Yaskawa INFORM job: DEMO_ROOF_UPPER_0625_3PAINT_41.JBI

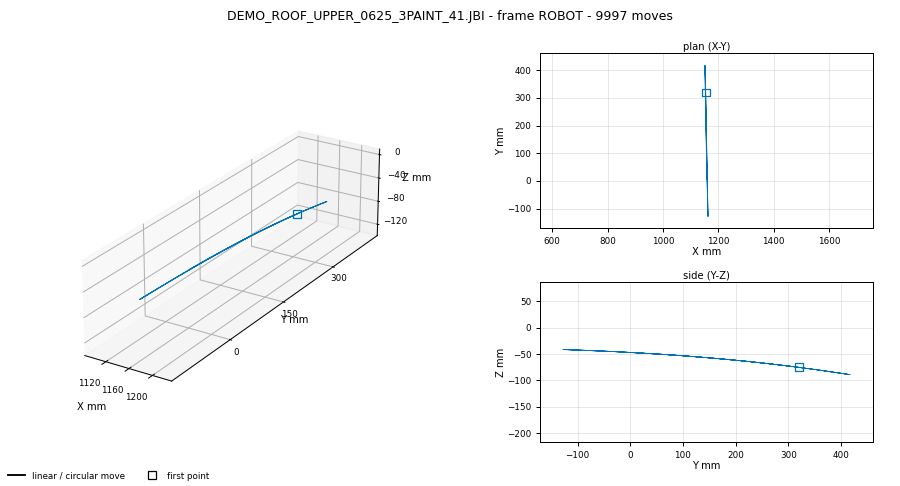
[picture p0: tool path of DEMO_ROOF_UPPER_0625_3PAINT_41.JBI in frame ROBOT, 9997 of 9997 moves have a stored position in this frame; points joined in program order, loops and branches not executed]
/JOB
//NAME DEMO_ROOF_UPPER_0625_3PAINT41
//POS
///NPOS 9997,0,0,0,0,0
///TOOL 0
///USER 0
///POSTYPE ROBOT
///RECTAN
///RCONF 1,0,0,0,0,0,0,0,0,0,0,0,0,0,0,0,0,0,0,0,0,0,0,0
C00000=1155.027,319.870,-75.171,-176.725,8.570,148.744
C00001=1155.032,319.622,-75.138,-176.728,8.567,148.744
C00002=1155.036,319.374,-75.107,-176.730,8.563,148.743
C00003=1155.040,319.126,-75.075,-176.733,8.560,148.743
C00004=1155.044,318.878,-75.042,-176.735,8.557,148.743
C00005=1155.048,318.630,-75.011,-176.738,8.553,148.743
C00006=1155.052,318.382,-74.979,-176.741,8.550,148.743
C00007=1155.057,318.134,-74.947,-176.743,8.546,148.743
C00008=1155.060,317.886,-74.915,-176.746,8.542,148.742
C00009=1155.065,317.639,-74.883,-176.748,8.539,148.742
C00010=1155.069,317.390,-74.851,-176.751,8.536,148.742
C00011=1155.073,317.142,-74.819,-176.753,8.533,148.742
C00012=1155.077,316.895,-74.788,-176.756,8.529,148.742
C00013=1155.081,316.647,-74.756,-176.758,8.525,148.742
C00014=1155.085,316.399,-74.723,-176.761,8.522,148.742
C00015=1155.090,316.151,-74.692,-176.764,8.519,148.742
C00016=1155.093,315.903,-74.660,-176.766,8.515,148.741
C00017=1155.097,315.655,-74.629,-176.769,8.512,148.741
C00018=1155.102,315.407,-74.597,-176.771,8.509,148.741
C00019=1155.106,315.159,-74.565,-176.774,8.506,148.741
C00020=1155.110,314.911,-74.533,-176.777,8.502,148.741
C00021=1155.114,314.663,-74.502,-176.779,8.499,148.741
C00022=1155.119,314.415,-74.469,-176.782,8.495,148.741
C00023=1155.123,314.167,-74.438,-176.784,8.492,148.740
C00024=1155.128,313.890,-74.403,-176.787,8.488,148.740
C00025=1155.132,313.612,-74.367,-176.790,8.484,148.740
C00026=1155.137,313.335,-74.332,-176.793,8.480,148.740
C00027=1155.141,313.058,-74.296,-176.795,8.477,148.740
C00028=1155.146,312.810,-74.265,-176.799,8.473,148.740
C00029=1155.149,312.562,-74.234,-176.801,8.470,148.739
C00030=1155.153,312.314,-74.202,-176.803,8.466,148.739
C00031=1155.159,312.065,-74.170,-176.806,8.463,148.739
C00032=1155.162,311.817,-74.139,-176.809,8.460,148.739
C00033=1155.167,311.570,-74.107,-176.811,8.456,148.739
C00034=1155.171,311.321,-74.076,-176.814,8.453,148.739
C00035=1155.175,311.074,-74.045,-176.816,8.450,148.739
C00036=1155.179,310.826,-74.013,-176.819,8.447,148.739
C00037=1155.183,310.578,-73.982,-176.822,8.443,148.739
C00038=1155.187,310.330,-73.950,-176.824,8.440,148.738
C00039=1155.191,310.082,-73.919,-176.827,8.436,148.738
C00040=1155.195,309.834,-73.887,-176.830,8.433,148.738
C00041=1155.200,309.586,-73.857,-176.832,8.430,148.738
C00042=1155.204,309.338,-73.825,-176.835,8.426,148.738
C00043=1155.208,309.090,-73.794,-176.837,8.423,148.738
C00044=1155.212,308.842,-73.762,-176.840,8.420,148.738
C00045=1155.216,308.594,-73.731,-176.842,8.416,148.737
C00046=1155.220,308.346,-73.700,-176.845,8.413,148.737
C00047=1155.225,308.098,-73.669,-176.848,8.409,148.737
C00048=1155.228,307.850,-73.637,-176.850,8.406,148.737
C00049=1155.233,307.602,-73.606,-176.853,8.403,148.737
C00050=1155.237,307.353,-73.575,-176.855,8.400,148.737
C00051=1155.241,307.106,-73.544,-176.858,8.397,148.737
C00052=1155.245,306.857,-73.513,-176.861,8.393,148.737
C00053=1155.250,306.610,-73.481,-176.863,8.389,148.736
C00054=1155.254,306.362,-73.450,-176.866,8.387,148.737
C00055=1155.258,306.114,-73.419,-176.868,8.383,148.736
C00056=1155.263,305.866,-73.388,-176.871,8.380,148.736
C00057=1155.267,305.618,-73.357,-176.874,8.376,148.736
C00058=1155.271,305.370,-73.326,-176.876,8.373,148.736
C00059=1155.275,305.121,-73.295,-176.879,8.370,148.736
C00060=1155.279,304.874,-73.264,-176.881,8.367,148.736
C00061=1155.283,304.626,-73.233,-176.884,8.364,148.736
C00062=1155.287,304.377,-73.202,-176.887,8.360,148.736
C00063=1155.292,304.129,-73.171,-176.889,8.356,148.735
C00064=1155.296,303.882,-73.140,-176.892,8.353,148.735
C00065=1155.300,303.633,-73.108,-176.894,8.350,148.735
C00066=1155.304,303.386,-73.078,-176.897,8.347,148.735
C00067=1155.308,303.137,-73.047,-176.899,8.344,148.735
C00068=1155.313,302.889,-73.016,-176.903,8.340,148.735
C00069=1155.317,302.642,-72.985,-176.905,8.337,148.735
C00070=1155.321,302.393,-72.954,-176.907,8.334,148.735
C00071=1155.325,302.145,-72.924,-176.910,8.331,148.735
C00072=1155.330,301.897,-72.893,-176.912,8.327,148.735
C00073=1155.334,301.649,-72.862,-176.915,8.324,148.735
C00074=1155.338,301.401,-72.831,-176.918,8.320,148.734
C00075=1155.342,301.153,-72.801,-176.921,8.317,148.734
C00076=1155.346,300.905,-72.770,-176.923,8.314,148.734
C00077=1155.351,300.657,-72.739,-176.926,8.311,148.734
C00078=1155.355,300.409,-72.708,-176.928,8.308,148.734
C00079=1155.359,300.161,-72.678,-176.931,8.305,148.734
C00080=1155.363,299.912,-72.647,-176.934,8.301,148.734
C00081=1155.368,299.664,-72.616,-176.937,8.298,148.734
C00082=1155.372,299.417,-72.586,-176.939,8.295,148.734
C00083=1155.376,299.168,-72.555,-176.941,8.291,148.734
C00084=1155.380,298.920,-72.524,-176.944,8.288,148.734
C00085=1155.384,298.672,-72.494,-176.946,8.285,148.733
C00086=1155.389,298.424,-72.463,-176.950,8.281,148.733
C00087=1155.393,298.176,-72.432,-176.952,8.278,148.733
C00088=1155.397,297.928,-72.402,-176.955,8.275,148.733
C00089=1155.402,297.680,-72.372,-176.957,8.272,148.733
C00090=1155.406,297.432,-72.342,-176.960,8.269,148.733
C00091=1155.410,297.183,-72.310,-176.962,8.266,148.733
C00092=1155.414,296.935,-72.280,-176.965,8.263,148.733
C00093=1155.418,296.688,-72.250,-176.968,8.259,148.733
C00094=1155.423,296.440,-72.219,-176.970,8.255,148.733
C00095=1155.426,296.191,-72.189,-176.973,8.253,148.733
C00096=1155.431,295.943,-72.158,-176.976,8.249,148.733
C00097=1155.435,295.695,-72.128,-176.978,8.246,148.733
C00098=1155.439,295.447,-72.097,-176.981,8.243,148.733
C00099=1155.444,295.199,-72.068,-176.983,8.240,148.733
C00100=1155.448,294.950,-72.037,-176.986,8.237,148.732
C00101=1155.452,294.703,-72.006,-176.989,8.233,148.732
C00102=1155.456,294.454,-71.976,-176.991,8.230,148.732
C00103=1155.460,294.206,-71.946,-176.994,8.227,148.732
C00104=1155.465,293.958,-71.916,-176.996,8.224,148.732
C00105=1155.468,293.709,-71.886,-176.999,8.221,148.732
C00106=1155.473,293.461,-71.855,-177.002,8.218,148.732
C00107=1155.477,293.214,-71.825,-177.004,8.214,148.732
C00108=1155.482,292.965,-71.795,-177.007,8.211,148.732
C00109=1155.486,292.718,-71.765,-177.010,8.207,148.732
C00110=1155.490,292.469,-71.735,-177.013,8.204,148.732
C00111=1155.495,292.221,-71.704,-177.015,8.201,148.732
C00112=1155.498,291.973,-71.674,-177.018,8.198,148.732
C00113=1155.503,291.724,-71.644,-177.020,8.195,148.732
C00114=1155.507,291.477,-71.614,-177.023,8.192,148.732
C00115=1155.511,291.229,-71.584,-177.026,8.189,148.732
C00116=1155.515,290.981,-71.553,-177.028,8.186,148.731
C00117=1155.520,290.732,-71.524,-177.031,8.183,148.731
C00118=1155.523,290.485,-71.494,-177.033,8.179,148.731
C00119=1155.528,290.236,-71.464,-177.036,8.176,148.731
C00120=1155.533,289.988,-71.434,-177.039,8.173,148.731
C00121=1155.536,289.739,-71.404,-177.041,8.169,148.731
C00122=1155.541,289.491,-71.374,-177.044,8.166,148.731
C00123=1155.545,289.243,-71.343,-177.046,8.163,148.731
C00124=1155.549,288.995,-71.314,-177.049,8.160,148.731
C00125=1155.554,288.746,-71.284,-177.052,8.157,148.731
C00126=1155.558,288.499,-71.254,-177.054,8.154,148.731
C00127=1155.562,288.251,-71.224,-177.057,8.151,148.731
C00128=1155.566,287.976,-71.191,-177.060,8.147,148.731
C00129=1155.571,287.700,-71.158,-177.063,8.144,148.731
C00130=1155.576,287.426,-71.125,-177.066,8.140,148.731
C00131=1155.580,287.149,-71.092,-177.069,8.137,148.731
C00132=1155.585,286.902,-71.061,-177.072,8.133,148.731
C00133=1155.589,286.653,-71.032,-177.074,8.130,148.731
C00134=1155.593,286.405,-71.002,-177.077,8.127,148.731
C00135=1155.598,286.157,-70.973,-177.080,8.124,148.731
C00136=1155.602,285.909,-70.942,-177.082,8.121,148.731
C00137=1155.606,285.661,-70.913,-177.085,8.118,148.731
C00138=1155.611,285.412,-70.883,-177.087,8.115,148.730
C00139=1155.615,285.164,-70.854,-177.090,8.112,148.730
C00140=1155.619,284.916,-70.825,-177.093,8.109,148.731
C00141=1155.624,284.668,-70.795,-177.095,8.106,148.730
C00142=1155.628,284.420,-70.765,-177.098,8.103,148.730
C00143=1155.632,284.172,-70.735,-177.101,8.100,148.730
C00144=1155.637,283.924,-70.706,-177.103,8.096,148.730
C00145=1155.641,283.675,-70.676,-177.106,8.094,148.730
C00146=1155.645,283.427,-70.647,-177.109,8.091,148.730
C00147=1155.649,283.179,-70.617,-177.111,8.086,148.730
C00148=1155.653,282.931,-70.588,-177.114,8.084,148.730
C00149=1155.658,282.682,-70.558,-177.117,8.081,148.730
C00150=1155.662,282.434,-70.529,-177.119,8.077,148.730
C00151=1155.666,282.186,-70.500,-177.122,8.074,148.730
C00152=1155.671,281.937,-70.469,-177.125,8.071,148.730
C00153=1155.675,281.689,-70.440,-177.128,8.068,148.730
C00154=1155.679,281.441,-70.411,-177.130,8.065,148.730
C00155=1155.684,281.193,-70.381,-177.133,8.062,148.730
C00156=1155.688,280.945,-70.352,-177.135,8.059,148.730
C00157=1155.692,280.697,-70.323,-177.138,8.056,148.730
C00158=1155.697,280.448,-70.293,-177.140,8.053,148.730
C00159=1155.701,280.200,-70.264,-177.143,8.050,148.730
C00160=1155.705,279.952,-70.234,-177.146,8.047,148.730
C00161=1155.709,279.703,-70.205,-177.148,8.044,148.730
C00162=1155.714,279.455,-70.176,-177.151,8.041,148.730
C00163=1155.718,279.207,-70.147,-177.154,8.038,148.730
C00164=1155.722,278.959,-70.118,-177.157,8.035,148.730
C00165=1155.726,278.711,-70.089,-177.159,8.032,148.730
C00166=1155.730,278.463,-70.059,-177.162,8.029,148.730
C00167=1155.735,278.214,-70.030,-177.164,8.026,148.730
C00168=1155.739,277.965,-70.001,-177.167,8.023,148.730
C00169=1155.744,277.718,-69.972,-177.170,8.020,148.730
C00170=1155.748,277.470,-69.942,-177.172,8.017,148.730
C00171=1155.752,277.221,-69.914,-177.175,8.014,148.730
C00172=1155.756,276.972,-69.884,-177.178,8.010,148.730
C00173=1155.761,276.724,-69.855,-177.181,8.007,148.730
C00174=1155.765,276.477,-69.826,-177.184,8.004,148.730
C00175=1155.769,276.228,-69.798,-177.186,8.001,148.730
C00176=1155.773,275.980,-69.768,-177.189,7.998,148.730
C00177=1155.778,275.731,-69.739,-177.191,7.995,148.730
C00178=1155.782,275.483,-69.710,-177.194,7.992,148.730
C00179=1155.787,275.235,-69.681,-177.197,7.989,148.730
C00180=1155.790,274.987,-69.652,-177.200,7.986,148.730
C00181=1155.795,274.738,-69.623,-177.202,7.983,148.730
C00182=1155.799,274.490,-69.594,-177.205,7.979,148.730
C00183=1155.804,274.242,-69.565,-177.207,7.977,148.730
C00184=1155.807,273.994,-69.537,-177.210,7.974,148.730
C00185=1155.812,273.745,-69.508,-177.213,7.971,148.730
C00186=1155.816,273.497,-69.478,-177.216,7.968,148.730
C00187=1155.821,273.248,-69.450,-177.218,7.964,148.730
C00188=1155.825,273.000,-69.421,-177.221,7.961,148.730
C00189=1155.829,272.752,-69.392,-177.224,7.959,148.730
C00190=1155.833,272.503,-69.363,-177.226,7.956,148.730
C00191=1155.838,272.255,-69.335,-177.229,7.953,148.730
C00192=1155.842,272.007,-69.306,-177.231,7.949,148.730
C00193=1155.846,271.758,-69.277,-177.234,7.946,148.730
C00194=1155.851,271.511,-69.248,-177.237,7.943,148.730
C00195=1155.855,271.262,-69.220,-177.240,7.941,148.730
C00196=1155.859,271.014,-69.190,-177.243,7.938,148.730
C00197=1155.864,270.766,-69.162,-177.245,7.935,148.730
C00198=1155.868,270.517,-69.134,-177.248,7.931,148.730
C00199=1155.872,270.269,-69.104,-177.250,7.928,148.730
C00200=1155.877,270.021,-69.076,-177.253,7.926,148.730
C00201=1155.881,269.772,-69.048,-177.255,7.923,148.730
C00202=1155.885,269.524,-69.018,-177.258,7.920,148.730
C00203=1155.890,269.276,-68.990,-177.261,7.917,148.730
C00204=1155.894,269.027,-68.962,-177.263,7.914,148.730
C00205=1155.899,268.779,-68.933,-177.266,7.911,148.730
C00206=1155.902,268.531,-68.905,-177.269,7.908,148.730
C00207=1155.907,268.282,-68.876,-177.272,7.905,148.730
C00208=1155.911,268.034,-68.848,-177.274,7.902,148.730
C00209=1155.916,267.785,-68.819,-177.277,7.899,148.730
C00210=1155.920,267.537,-68.790,-177.280,7.896,148.730
C00211=1155.924,267.289,-68.762,-177.283,7.894,148.731
C00212=1155.929,267.040,-68.733,-177.285,7.890,148.730
C00213=1155.933,266.792,-68.706,-177.288,7.887,148.730
C00214=1155.938,266.543,-68.677,-177.290,7.884,148.730
C00215=1155.942,266.296,-68.648,-177.293,7.881,148.731
C00216=1155.946,266.047,-68.620,-177.296,7.878,148.731
C00217=1155.950,265.799,-68.591,-177.299,7.876,148.731
C00218=1155.955,265.551,-68.563,-177.302,7.873,148.731
C00219=1155.959,265.302,-68.535,-177.304,7.870,148.731
C00220=1155.964,265.054,-68.507,-177.307,7.867,148.731
C00221=1155.968,264.805,-68.478,-177.309,7.863,148.731
C00222=1155.973,264.557,-68.450,-177.312,7.860,148.731
C00223=1155.976,264.308,-68.422,-177.315,7.858,148.731
C00224=1155.981,264.061,-68.394,-177.318,7.855,148.731
C00225=1155.985,263.812,-68.365,-177.320,7.852,148.731
C00226=1155.990,263.564,-68.338,-177.323,7.850,148.731
C00227=1155.994,263.315,-68.309,-177.325,7.847,148.731
C00228=1155.998,263.067,-68.281,-177.328,7.844,148.731
C00229=1156.002,262.818,-68.253,-177.331,7.841,148.731
C00230=1156.007,262.570,-68.225,-177.334,7.838,148.731
C00231=1156.011,262.322,-68.196,-177.336,7.835,148.731
C00232=1156.016,262.048,-68.166,-177.339,7.832,148.731
C00233=1156.021,261.775,-68.135,-177.343,7.828,148.731
C00234=1156.026,261.501,-68.104,-177.345,7.825,148.731
C00235=1156.030,261.229,-68.072,-177.348,7.822,148.731
C00236=1156.035,260.980,-68.045,-177.351,7.819,148.732
C00237=1156.039,260.731,-68.017,-177.354,7.816,148.732
C00238=1156.044,260.483,-67.989,-177.356,7.813,148.732
C00239=1156.047,260.235,-67.961,-177.359,7.810,148.732
C00240=1156.052,259.987,-67.933,-177.362,7.807,148.732
C00241=1156.057,259.738,-67.905,-177.365,7.805,148.732
C00242=1156.061,259.490,-67.877,-177.368,7.802,148.732
C00243=1156.065,259.242,-67.849,-177.370,7.798,148.732
C00244=1156.069,258.993,-67.821,-177.373,7.795,148.732
C00245=1156.074,258.745,-67.793,-177.375,7.792,148.732
C00246=1156.078,258.496,-67.765,-177.378,7.790,148.732
C00247=1156.082,258.248,-67.738,-177.380,7.787,148.732
C00248=1156.087,258.000,-67.710,-177.383,7.784,148.732
C00249=1156.092,257.750,-67.682,-177.386,7.781,148.732
C00250=1156.096,257.503,-67.654,-177.389,7.779,148.732
C00251=1156.100,257.254,-67.626,-177.391,7.776,148.732
C00252=1156.104,257.006,-67.599,-177.394,7.773,148.732
C00253=1156.109,256.758,-67.571,-177.397,7.770,148.732
C00254=1156.113,256.509,-67.542,-177.400,7.767,148.732
C00255=1156.118,256.260,-67.515,-177.403,7.764,148.732
C00256=1156.122,256.012,-67.488,-177.405,7.762,148.733
C00257=1156.126,255.763,-67.460,-177.407,7.759,148.733
C00258=1156.131,255.515,-67.432,-177.410,7.756,148.733
C00259=1156.135,255.267,-67.405,-177.413,7.753,148.733
C00260=1156.139,255.018,-67.377,-177.416,7.750,148.733
C00261=1156.144,254.770,-67.350,-177.419,7.747,148.733
C00262=1156.149,254.522,-67.322,-177.421,7.744,148.733
C00263=1156.153,254.273,-67.294,-177.424,7.741,148.733
C00264=1156.157,254.025,-67.266,-177.427,7.738,148.733
C00265=1156.162,253.776,-67.239,-177.429,7.736,148.733
C00266=1156.166,253.527,-67.211,-177.432,7.733,148.733
C00267=1156.170,253.279,-67.184,-177.435,7.730,148.734
C00268=1156.175,253.031,-67.156,-177.438,7.728,148.734
C00269=1156.179,252.783,-67.129,-177.441,7.725,148.734
C00270=1156.183,252.534,-67.101,-177.443,7.722,148.734
C00271=1156.188,252.286,-67.074,-177.446,7.719,148.734
C00272=1156.192,252.037,-67.047,-177.449,7.716,148.734
C00273=1156.196,251.788,-67.019,-177.451,7.714,148.734
C00274=1156.201,251.540,-66.992,-177.454,7.711,148.734
C00275=1156.205,251.291,-66.965,-177.457,7.708,148.734
C00276=1156.210,251.044,-66.937,-177.459,7.705,148.734
C00277=1156.214,250.794,-66.910,-177.462,7.702,148.734
C00278=1156.218,250.546,-66.883,-177.465,7.699,148.734
C00279=1156.223,250.298,-66.855,-177.468,7.696,148.734
C00280=1156.227,250.050,-66.828,-177.470,7.694,148.734
C00281=1156.232,249.800,-66.800,-177.473,7.691,148.735
C00282=1156.236,249.552,-66.773,-177.476,7.688,148.735
C00283=1156.240,249.304,-66.746,-177.478,7.685,148.735
C00284=1156.244,249.056,-66.719,-177.482,7.682,148.735
C00285=1156.249,248.807,-66.692,-177.484,7.680,148.735
C00286=1156.253,248.558,-66.665,-177.487,7.677,148.735
C00287=1156.258,248.310,-66.637,-177.489,7.674,148.735
C00288=1156.262,248.062,-66.610,-177.492,7.672,148.735
C00289=1156.267,247.813,-66.583,-177.495,7.669,148.735
C00290=1156.271,247.565,-66.556,-177.498,7.666,148.735
C00291=1156.275,247.317,-66.529,-177.500,7.663,148.735
C00292=1156.279,247.067,-66.502,-177.503,7.660,148.736
C00293=1156.284,246.819,-66.475,-177.505,7.658,148.736
C00294=1156.289,246.570,-66.448,-177.508,7.655,148.736
C00295=1156.293,246.322,-66.420,-177.511,7.652,148.736
C00296=1156.298,246.073,-66.393,-177.514,7.649,148.736
C00297=1156.302,245.826,-66.366,-177.517,7.646,148.736
C00298=1156.306,245.577,-66.339,-177.520,7.643,148.736
C00299=1156.310,245.328,-66.312,-177.522,7.641,148.736
C00300=1156.315,245.080,-66.285,-177.525,7.638,148.736
C00301=1156.319,244.831,-66.258,-177.527,7.635,148.736
C00302=1156.324,244.583,-66.231,-177.530,7.632,148.737
C00303=1156.328,244.334,-66.204,-177.533,7.630,148.737
C00304=1156.333,244.086,-66.177,-177.536,7.628,148.737
C00305=1156.337,243.837,-66.151,-177.538,7.625,148.737
C00306=1156.342,243.589,-66.124,-177.541,7.622,148.737
C00307=1156.346,243.340,-66.097,-177.544,7.619,148.737
C00308=1156.350,243.091,-66.070,-177.547,7.616,148.737
C00309=1156.354,242.843,-66.043,-177.549,7.614,148.737
C00310=1156.359,242.594,-66.016,-177.552,7.611,148.737
C00311=1156.364,242.346,-65.989,-177.555,7.608,148.738
C00312=1156.368,242.098,-65.963,-177.558,7.605,148.738
C00313=1156.372,241.849,-65.936,-177.560,7.602,148.738
C00314=1156.377,241.600,-65.910,-177.563,7.600,148.738
C00315=1156.381,241.352,-65.883,-177.565,7.597,148.738
C00316=1156.386,241.103,-65.856,-177.568,7.594,148.738
C00317=1156.390,240.855,-65.829,-177.571,7.592,148.738
C00318=1156.394,240.607,-65.802,-177.574,7.589,148.738
C00319=1156.399,240.357,-65.776,-177.576,7.587,148.739
C00320=1156.403,240.109,-65.749,-177.579,7.584,148.739
C00321=1156.408,239.861,-65.722,-177.582,7.581,148.739
C00322=1156.412,239.612,-65.697,-177.585,7.578,148.739
C00323=1156.417,239.363,-65.670,-177.588,7.575,148.739
C00324=1156.422,239.115,-65.642,-177.590,7.573,148.739
C00325=1156.425,238.867,-65.616,-177.593,7.570,148.739
C00326=1156.430,238.618,-65.590,-177.596,7.567,148.739
C00327=1156.434,238.370,-65.563,-177.599,7.564,148.739
C00328=1156.439,238.121,-65.536,-177.601,7.563,148.740
C00329=1156.443,237.872,-65.510,-177.604,7.560,148.740
C00330=1156.448,237.624,-65.483,-177.607,7.557,148.740
C00331=1156.452,237.375,-65.458,-177.610,7.554,148.740
C00332=1156.457,237.126,-65.431,-177.612,7.552,148.740
C00333=1156.461,236.878,-65.404,-177.615,7.549,148.740
C00334=1156.466,236.629,-65.378,-177.618,7.546,148.740
C00335=1156.470,236.381,-65.351,-177.621,7.543,148.741
C00336=1156.475,236.109,-65.323,-177.623,7.540,148.741
C00337=1156.479,235.837,-65.294,-177.627,7.538,148.741
C00338=1156.484,235.566,-65.264,-177.629,7.535,148.741
C00339=1156.489,235.294,-65.236,-177.632,7.532,148.741
C00340=1156.494,235.045,-65.209,-177.635,7.529,148.741
C00341=1156.498,234.797,-65.184,-177.638,7.526,148.741
C00342=1156.502,234.548,-65.157,-177.640,7.524,148.742
C00343=1156.507,234.299,-65.131,-177.643,7.521,148.742
C00344=1156.512,234.051,-65.105,-177.646,7.518,148.742
C00345=1156.516,233.803,-65.078,-177.649,7.516,148.742
C00346=1156.521,233.554,-65.053,-177.651,7.514,148.742
C00347=1156.525,233.306,-65.026,-177.654,7.511,148.742
C00348=1156.530,233.057,-65.000,-177.657,7.508,148.742
C00349=1156.534,232.808,-64.974,-177.660,7.505,148.743
C00350=1156.538,232.560,-64.948,-177.662,7.503,148.743
C00351=1156.543,232.311,-64.921,-177.665,7.500,148.743
C00352=1156.547,232.062,-64.896,-177.668,7.497,148.743
C00353=1156.551,231.814,-64.869,-177.671,7.494,148.743
C00354=1156.556,231.565,-64.843,-177.673,7.492,148.743
C00355=1156.561,231.316,-64.817,-177.676,7.489,148.743
C00356=1156.564,231.068,-64.791,-177.679,7.486,148.743
C00357=1156.570,230.820,-64.765,-177.682,7.485,148.744
C00358=1156.574,230.571,-64.739,-177.684,7.482,148.744
C00359=1156.579,230.322,-64.713,-177.687,7.479,148.744
C00360=1156.582,230.074,-64.687,-177.690,7.476,148.744
C00361=1156.587,229.825,-64.661,-177.693,7.474,148.744
C00362=1156.592,229.576,-64.635,-177.695,7.471,148.744
C00363=1156.596,229.328,-64.609,-177.698,7.468,148.744
C00364=1156.601,229.079,-64.584,-177.701,7.466,148.745
C00365=1156.605,228.830,-64.558,-177.704,7.464,148.745
C00366=1156.610,228.582,-64.531,-177.706,7.461,148.745
C00367=1156.614,228.334,-64.505,-177.709,7.458,148.745
C00368=1156.619,228.085,-64.480,-177.712,7.456,148.745
C00369=1156.623,227.836,-64.454,-177.715,7.453,148.745
C00370=1156.627,227.587,-64.428,-177.717,7.450,148.746
C00371=1156.633,227.339,-64.402,-177.720,7.448,148.746
C00372=1156.637,227.090,-64.376,-177.723,7.445,148.746
C00373=1156.641,226.841,-64.351,-177.726,7.442,148.746
C00374=1156.645,226.592,-64.325,-177.728,7.441,148.746
C00375=1156.650,226.344,-64.300,-177.731,7.438,148.746
C00376=1156.654,226.096,-64.274,-177.734,7.435,148.747
C00377=1156.659,225.847,-64.248,-177.736,7.433,148.747
C00378=1156.663,225.599,-64.223,-177.739,7.430,148.747
C00379=1156.668,225.350,-64.196,-177.742,7.427,148.747
C00380=1156.673,225.101,-64.171,-177.744,7.425,148.747
C00381=1156.677,224.852,-64.145,-177.747,7.422,148.747
C00382=1156.682,224.604,-64.119,-177.750,7.419,148.748
C00383=1156.686,224.355,-64.094,-177.752,7.417,148.748
C00384=1156.690,224.106,-64.068,-177.756,7.415,148.748
C00385=1156.695,223.858,-64.043,-177.758,7.412,148.748
C00386=1156.699,223.609,-64.017,-177.761,7.410,148.748
C00387=1156.703,223.360,-63.991,-177.764,7.407,148.749
C00388=1156.708,223.112,-63.966,-177.767,7.404,148.749
C00389=1156.713,222.863,-63.941,-177.769,7.402,148.749
C00390=1156.717,222.614,-63.915,-177.772,7.399,148.749
C00391=1156.722,222.366,-63.890,-177.775,7.397,148.749
C00392=1156.726,222.117,-63.864,-177.777,7.394,148.749
C00393=1156.731,221.869,-63.838,-177.780,7.392,148.750
C00394=1156.735,221.620,-63.813,-177.783,7.389,148.750
C00395=1156.740,221.371,-63.788,-177.786,7.387,148.750
C00396=1156.744,221.123,-63.762,-177.789,7.384,148.750
C00397=1156.749,220.874,-63.736,-177.791,7.381,148.750
C00398=1156.753,220.625,-63.711,-177.794,7.380,148.750
C00399=1156.758,220.376,-63.686,-177.797,7.377,148.751
C00400=1156.762,220.128,-63.660,-177.799,7.374,148.751
C00401=1156.766,219.880,-63.635,-177.802,7.372,148.751
C00402=1156.771,219.630,-63.610,-177.805,7.369,148.751
C00403=1156.775,219.382,-63.585,-177.807,7.367,148.751
C00404=1156.780,219.134,-63.559,-177.811,7.364,148.751
C00405=1156.784,218.884,-63.534,-177.813,7.361,148.752
C00406=1156.789,218.636,-63.509,-177.816,7.360,148.752
C00407=1156.793,218.387,-63.483,-177.819,7.357,148.752
C00408=1156.799,218.138,-63.458,-177.821,7.355,148.752
C00409=1156.802,217.890,-63.433,-177.824,7.352,148.752
C00410=1156.807,217.641,-63.409,-177.827,7.349,148.753
C00411=1156.811,217.392,-63.383,-177.829,7.347,148.753
C00412=1156.816,217.144,-63.357,-177.832,7.344,148.753
C00413=1156.821,216.895,-63.332,-177.835,7.341,148.753
C00414=1156.824,216.646,-63.307,-177.838,7.340,148.753
C00415=1156.829,216.398,-63.283,-177.841,7.337,148.753
C00416=1156.834,216.149,-63.257,-177.843,7.335,148.754
C00417=1156.839,215.900,-63.232,-177.846,7.332,148.754
C00418=1156.843,215.651,-63.206,-177.849,7.329,148.754
C00419=1156.847,215.403,-63.182,-177.852,7.327,148.754
C00420=1156.852,215.154,-63.157,-177.854,7.324,148.754
C00421=1156.857,214.905,-63.132,-177.857,7.322,148.755
C00422=1156.861,214.656,-63.108,-177.860,7.320,148.755
C00423=1156.865,214.408,-63.082,-177.862,7.318,148.755
C00424=1156.870,214.159,-63.057,-177.865,7.315,148.755
C00425=1156.875,213.911,-63.032,-177.868,7.312,148.755
C00426=1156.879,213.662,-63.008,-177.871,7.310,148.756
C00427=1156.884,213.413,-62.983,-177.874,7.307,148.756
C00428=1156.888,213.165,-62.957,-177.876,7.305,148.756
C00429=1156.892,212.916,-62.933,-177.879,7.303,148.756
C00430=1156.897,212.668,-62.907,-177.882,7.300,148.756
C00431=1156.902,212.418,-62.882,-177.885,7.298,148.757
C00432=1156.906,212.170,-62.858,-177.887,7.295,148.757
C00433=1156.911,211.920,-62.833,-177.890,7.293,148.757
C00434=1156.915,211.672,-62.808,-177.893,7.290,148.757
C00435=1156.920,211.424,-62.784,-177.895,7.288,148.757
C00436=1156.924,211.174,-62.759,-177.898,7.286,148.758
C00437=1156.928,210.927,-62.734,-177.900,7.283,148.758
C00438=1156.933,210.677,-62.709,-177.904,7.281,148.758
C00439=1156.938,210.428,-62.684,-177.906,7.278,148.758
C00440=1156.943,210.158,-62.658,-177.909,7.276,148.759
C00441=1156.948,209.887,-62.631,-177.912,7.273,148.759
C00442=1156.953,209.617,-62.604,-177.915,7.271,148.759
C00443=1156.957,209.346,-62.577,-177.918,7.268,148.759
C00444=1156.962,209.098,-62.553,-177.921,7.265,148.759
C00445=1156.967,208.849,-62.528,-177.924,7.263,148.760
C00446=1156.971,208.600,-62.504,-177.927,7.261,148.760
C00447=1156.976,208.351,-62.479,-177.929,7.259,148.760
C00448=1156.980,208.102,-62.454,-177.932,7.256,148.760
C00449=1156.985,207.853,-62.430,-177.934,7.254,148.760
C00450=1156.990,207.605,-62.404,-177.938,7.251,148.761
C00451=1156.993,207.356,-62.380,-177.940,7.249,148.761
C00452=1156.999,207.108,-62.355,-177.943,7.246,148.761
C00453=1157.003,206.859,-62.331,-177.945,7.244,148.761
C00454=1157.007,206.611,-62.307,-177.949,7.242,148.762
C00455=1157.012,206.361,-62.282,-177.951,7.239,148.762
C00456=1157.016,206.113,-62.258,-177.954,7.237,148.762
C00457=1157.021,205.864,-62.233,-177.957,7.234,148.762
C00458=1157.025,205.615,-62.209,-177.959,7.232,148.763
C00459=1157.030,205.366,-62.184,-177.962,7.229,148.763
C00460=1157.035,205.118,-62.160,-177.965,7.228,148.763
C00461=1157.040,204.869,-62.135,-177.968,7.225,148.763
C00462=1157.044,204.620,-62.111,-177.970,7.223,148.763
C00463=1157.048,204.371,-62.088,-177.973,7.220,148.764
C00464=1157.053,204.122,-62.063,-177.976,7.218,148.764
C00465=1157.057,203.873,-62.039,-177.979,7.215,148.764
C00466=1157.062,203.625,-62.014,-177.981,7.214,148.764
C00467=1157.067,203.376,-61.990,-177.984,7.211,148.764
C00468=1157.071,203.128,-61.966,-177.987,7.209,148.765
C00469=1157.075,202.879,-61.941,-177.990,7.206,148.765
C00470=1157.080,202.630,-61.917,-177.992,7.204,148.765
C00471=1157.085,202.381,-61.893,-177.995,7.202,148.766
C00472=1157.089,202.132,-61.869,-177.998,7.200,148.766
C00473=1157.094,201.884,-61.845,-178.001,7.197,148.766
C00474=1157.098,201.635,-61.820,-178.003,7.195,148.766
C00475=1157.103,201.386,-61.796,-178.006,7.192,148.766
C00476=1157.108,201.137,-61.772,-178.009,7.190,148.767
C00477=1157.112,200.888,-61.748,-178.012,7.188,148.767
C00478=1157.117,200.640,-61.724,-178.014,7.185,148.767
C00479=1157.121,200.391,-61.699,-178.017,7.183,148.767
C00480=1157.126,200.141,-61.676,-178.020,7.181,148.767
C00481=1157.130,199.893,-61.651,-178.023,7.178,148.768
C00482=1157.135,199.645,-61.627,-178.025,7.176,148.768
C00483=1157.139,199.396,-61.604,-178.028,7.174,148.768
C00484=1157.145,199.147,-61.579,-178.031,7.172,148.769
C00485=1157.148,198.898,-61.555,-178.033,7.170,148.769
C00486=1157.153,198.649,-61.532,-178.036,7.167,148.769
C00487=1157.157,198.400,-61.507,-178.039,7.165,148.769
C00488=1157.162,198.152,-61.483,-178.042,7.162,148.770
C00489=1157.167,197.903,-61.459,-178.044,7.160,148.770
C00490=1157.172,197.654,-61.435,-178.047,7.158,148.770
C00491=1157.176,197.405,-61.412,-178.050,7.156,148.770
C00492=1157.180,197.156,-61.388,-178.053,7.153,148.770
C00493=1157.185,196.907,-61.364,-178.056,7.151,148.771
C00494=1157.189,196.659,-61.340,-178.058,7.148,148.771
C00495=1157.194,196.410,-61.317,-178.061,7.147,148.771
C00496=1157.199,196.161,-61.292,-178.063,7.145,148.771
C00497=1157.204,195.912,-61.269,-178.066,7.142,148.772
C00498=1157.208,195.663,-61.245,-178.069,7.140,148.772
C00499=1157.213,195.414,-61.221,-178.072,7.137,148.772
C00500=1157.217,195.166,-61.197,-178.075,7.135,148.773
C00501=1157.222,194.917,-61.174,-178.077,7.133,148.773
C00502=1157.226,194.669,-61.150,-178.080,7.131,148.773
C00503=1157.231,194.419,-61.126,-178.083,7.128,148.773
C00504=1157.235,194.170,-61.102,-178.086,7.126,148.773
C00505=1157.240,193.921,-61.079,-178.088,7.124,148.774
C00506=1157.244,193.672,-61.055,-178.091,7.121,148.774
C00507=1157.249,193.424,-61.031,-178.094,7.120,148.774
C00508=1157.253,193.175,-61.008,-178.097,7.117,148.775
C00509=1157.258,192.926,-60.984,-178.099,7.115,148.775
C00510=1157.262,192.677,-60.960,-178.102,7.112,148.775
C00511=1157.267,192.428,-60.937,-178.105,7.110,148.775
C00512=1157.272,192.180,-60.913,-178.107,7.109,148.776
C00513=1157.276,191.931,-60.890,-178.111,7.106,148.776
C00514=1157.281,191.682,-60.866,-178.113,7.104,148.776
C00515=1157.286,191.433,-60.843,-178.116,7.101,148.776
C00516=1157.290,191.184,-60.819,-178.119,7.100,148.777
C00517=1157.295,190.935,-60.795,-178.121,7.097,148.777
C00518=1157.299,190.686,-60.772,-178.124,7.095,148.777
C00519=1157.304,190.437,-60.749,-178.126,7.093,148.777
C00520=1157.309,190.189,-60.725,-178.130,7.090,148.778
C00521=1157.313,189.940,-60.701,-178.132,7.088,148.778
C00522=1157.318,189.691,-60.678,-178.135,7.086,148.778
C00523=1157.323,189.442,-60.655,-178.138,7.084,148.778
C00524=1157.327,189.193,-60.631,-178.141,7.082,148.779
C00525=1157.332,188.944,-60.607,-178.143,7.079,148.779
C00526=1157.337,188.696,-60.584,-178.146,7.077,148.779
C00527=1157.341,188.447,-60.561,-178.149,7.076,148.780
C00528=1157.346,188.198,-60.538,-178.152,7.073,148.780
C00529=1157.350,187.949,-60.515,-178.154,7.071,148.780
C00530=1157.355,187.700,-60.491,-178.158,7.068,148.780
C00531=1157.360,187.451,-60.468,-178.160,7.066,148.781
C00532=1157.365,187.202,-60.445,-178.162,7.065,148.781
C00533=1157.369,186.953,-60.421,-178.166,7.062,148.781
C00534=1157.373,186.704,-60.399,-178.168,7.060,148.781
C00535=1157.378,186.456,-60.374,-178.171,7.057,148.782
C00536=1157.382,186.207,-60.351,-178.174,7.056,148.782
C00537=1157.387,185.958,-60.328,-178.176,7.053,148.782
C00538=1157.392,185.710,-60.305,-178.179,7.051,148.783
C00539=1157.396,185.461,-60.282,-178.182,7.049,148.783
C00540=1157.401,185.212,-60.259,-178.184,7.047,148.783
C00541=1157.406,184.963,-60.235,-178.187,7.044,148.783
C00542=1157.411,184.713,-60.213,-178.190,7.043,148.784
C00543=1157.415,184.464,-60.190,-178.192,7.041,148.784
C00544=1157.420,184.195,-60.164,-178.196,7.038,148.784
C00545=1157.425,183.926,-60.139,-178.199,7.035,148.785
C00546=1157.430,183.656,-60.115,-178.202,7.034,148.785
C00547=1157.435,183.386,-60.090,-178.205,7.031,148.785
C00548=1157.440,183.137,-60.066,-178.207,7.029,148.785
C00549=1157.444,182.888,-60.043,-178.210,7.026,148.786
C00550=1157.448,182.640,-60.020,-178.213,7.025,148.786
C00551=1157.454,182.391,-59.997,-178.215,7.023,148.786
C00552=1157.459,182.142,-59.974,-178.219,7.020,148.787
C00553=1157.462,181.893,-59.952,-178.221,7.018,148.787
C00554=1157.467,181.644,-59.928,-178.224,7.017,148.787
C00555=1157.471,181.395,-59.906,-178.227,7.014,148.787
C00556=1157.476,181.147,-59.883,-178.229,7.012,148.788
C00557=1157.481,180.897,-59.860,-178.232,7.010,148.788
C00558=1157.485,180.648,-59.837,-178.235,7.007,148.788
C00559=1157.490,180.399,-59.814,-178.238,7.005,148.789
C00560=1157.495,180.150,-59.790,-178.240,7.004,148.789
C00561=1157.500,179.902,-59.769,-178.244,7.001,148.789
C00562=1157.504,179.653,-59.745,-178.246,6.999,148.789
C00563=1157.508,179.404,-59.723,-178.248,6.997,148.790
C00564=1157.513,179.154,-59.700,-178.252,6.995,148.790
C00565=1157.518,178.906,-59.678,-178.254,6.993,148.790
C00566=1157.523,178.657,-59.654,-178.257,6.991,148.791
C00567=1157.527,178.408,-59.632,-178.260,6.988,148.791
C00568=1157.532,178.159,-59.609,-178.263,6.987,148.791
C00569=1157.537,177.911,-59.586,-178.265,6.984,148.792
C00570=1157.541,177.661,-59.564,-178.268,6.982,148.792
C00571=1157.546,177.412,-59.540,-178.271,6.980,148.792
C00572=1157.550,177.164,-59.518,-178.273,6.978,148.793
C00573=1157.555,176.914,-59.495,-178.276,6.975,148.793
C00574=1157.559,176.666,-59.473,-178.279,6.974,148.793
C00575=1157.564,176.416,-59.450,-178.282,6.972,148.793
C00576=1157.569,176.168,-59.428,-178.284,6.970,148.794
C00577=1157.574,175.918,-59.405,-178.287,6.967,148.794
C00578=1157.578,175.670,-59.382,-178.290,6.966,148.794
C00579=1157.583,175.421,-59.361,-178.292,6.964,148.795
C00580=1157.587,175.172,-59.337,-178.296,6.961,148.795
C00581=1157.592,174.923,-59.315,-178.298,6.959,148.795
C00582=1157.597,174.674,-59.292,-178.301,6.957,148.796
C00583=1157.601,174.425,-59.270,-178.304,6.955,148.796
C00584=1157.606,174.176,-59.247,-178.307,6.953,148.796
C00585=1157.611,173.927,-59.225,-178.309,6.951,148.797
C00586=1157.615,173.679,-59.202,-178.312,6.949,148.797
C00587=1157.620,173.429,-59.180,-178.315,6.947,148.797
C00588=1157.624,173.181,-59.157,-178.317,6.945,148.797
C00589=1157.629,172.931,-59.135,-178.320,6.943,148.798
C00590=1157.634,172.683,-59.113,-178.322,6.941,148.798
C00591=1157.638,172.434,-59.090,-178.326,6.939,148.798
C00592=1157.643,172.184,-59.067,-178.328,6.937,148.799
C00593=1157.648,171.936,-59.046,-178.331,6.935,148.799
C00594=1157.652,171.687,-59.023,-178.334,6.933,148.799
C00595=1157.658,171.438,-59.001,-178.337,6.930,148.800
C00596=1157.662,171.189,-58.979,-178.339,6.929,148.800
C00597=1157.666,170.940,-58.956,-178.342,6.927,148.800
C00598=1157.672,170.691,-58.934,-178.345,6.924,148.801
C00599=1157.676,170.442,-58.912,-178.348,6.923,148.801
C00600=1157.681,170.193,-58.890,-178.350,6.921,148.801
C00601=1157.685,169.944,-58.867,-178.353,6.919,148.802
C00602=1157.690,169.695,-58.845,-178.356,6.916,148.802
C00603=1157.695,169.446,-58.823,-178.359,6.914,148.802
C00604=1157.699,169.197,-58.801,-178.361,6.913,148.803
C00605=1157.704,168.948,-58.778,-178.364,6.911,148.803
C00606=1157.708,168.699,-58.756,-178.367,6.908,148.803
C00607=1157.713,168.450,-58.734,-178.370,6.906,148.804
C00608=1157.717,168.201,-58.712,-178.372,6.905,148.804
C00609=1157.722,167.952,-58.690,-178.375,6.903,148.804
C00610=1157.727,167.703,-58.668,-178.378,6.900,148.804
C00611=1157.732,167.455,-58.645,-178.381,6.898,148.805
C00612=1157.736,167.205,-58.623,-178.383,6.896,148.805
C00613=1157.741,166.957,-58.602,-178.386,6.895,148.805
C00614=1157.745,166.707,-58.580,-178.389,6.893,148.806
C00615=1157.751,166.458,-58.557,-178.392,6.890,148.806
C00616=1157.755,166.209,-58.535,-178.394,6.888,148.806
C00617=1157.760,165.960,-58.514,-178.397,6.887,148.807
C00618=1157.764,165.711,-58.491,-178.400,6.885,148.807
C00619=1157.769,165.462,-58.470,-178.403,6.882,148.807
C00620=1157.773,165.213,-58.448,-178.405,6.881,148.808
C00621=1157.778,164.964,-58.426,-178.408,6.879,148.808
C00622=1157.783,164.715,-58.403,-178.410,6.877,148.808
C00623=1157.788,164.466,-58.382,-178.413,6.875,148.809
C00624=1157.793,164.218,-58.360,-178.416,6.872,148.809
C00625=1157.797,163.968,-58.338,-178.419,6.871,148.809
C00626=1157.802,163.720,-58.316,-178.422,6.869,148.810
C00627=1157.806,163.470,-58.294,-178.424,6.867,148.810
C00628=1157.811,163.222,-58.273,-178.427,6.865,148.811
C00629=1157.816,162.972,-58.251,-178.430,6.863,148.811
C00630=1157.821,162.724,-58.229,-178.433,6.861,148.811
C00631=1157.825,162.475,-58.207,-178.435,6.859,148.811
C00632=1157.830,162.226,-58.185,-178.438,6.857,148.812
C00633=1157.835,161.977,-58.163,-178.441,6.856,148.812
C00634=1157.839,161.728,-58.141,-178.444,6.853,148.813
C00635=1157.844,161.478,-58.120,-178.447,6.851,148.813
C00636=1157.848,161.229,-58.098,-178.449,6.850,148.813
C00637=1157.853,160.980,-58.077,-178.452,6.847,148.813
C00638=1157.858,160.732,-58.055,-178.454,6.846,148.814
C00639=1157.862,160.482,-58.033,-178.458,6.843,148.814
C00640=1157.867,160.234,-58.011,-178.460,6.841,148.815
C00641=1157.872,159.984,-57.990,-178.463,6.840,148.815
C00642=1157.877,159.735,-57.968,-178.466,6.838,148.815
C00643=1157.881,159.487,-57.947,-178.468,6.836,148.816
C00644=1157.886,159.238,-57.925,-178.471,6.834,148.816
C00645=1157.891,158.988,-57.904,-178.474,6.832,148.816
C00646=1157.896,158.739,-57.882,-178.477,6.830,148.817
C00647=1157.900,158.490,-57.860,-178.479,6.828,148.817
C00648=1157.905,158.222,-57.837,-178.482,6.826,148.817
C00649=1157.911,157.952,-57.814,-178.485,6.824,148.818
C00650=1157.915,157.684,-57.791,-178.488,6.822,148.818
C00651=1157.921,157.414,-57.767,-178.491,6.820,148.818
C00652=1157.925,157.165,-57.745,-178.494,6.818,148.819
C00653=1157.930,156.916,-57.724,-178.497,6.816,148.819
C00654=1157.934,156.667,-57.703,-178.499,6.814,148.820
C00655=1157.939,156.419,-57.681,-178.502,6.813,148.820
C00656=1157.944,156.169,-57.660,-178.505,6.811,148.820
C00657=1157.949,155.920,-57.638,-178.508,6.808,148.821
C00658=1157.954,155.671,-57.617,-178.511,6.807,148.821
C00659=1157.958,155.422,-57.595,-178.513,6.805,148.821
C00660=1157.962,155.173,-57.574,-178.516,6.803,148.822
C00661=1157.967,154.924,-57.553,-178.519,6.801,148.822
C00662=1157.972,154.675,-57.532,-178.521,6.799,148.822
C00663=1157.977,154.425,-57.510,-178.524,6.798,148.823
C00664=1157.982,154.177,-57.489,-178.527,6.795,148.823
C00665=1157.986,153.928,-57.468,-178.530,6.793,148.823
C00666=1157.991,153.679,-57.447,-178.532,6.792,148.824
C00667=1157.996,153.429,-57.425,-178.535,6.790,148.824
C00668=1158.000,153.181,-57.404,-178.538,6.788,148.825
C00669=1158.006,152.931,-57.383,-178.541,6.786,148.825
C00670=1158.010,152.683,-57.362,-178.543,6.785,148.825
C00671=1158.015,152.434,-57.341,-178.546,6.783,148.826
C00672=1158.019,152.184,-57.319,-178.549,6.780,148.826
C00673=1158.024,151.935,-57.298,-178.552,6.779,148.826
C00674=1158.029,151.686,-57.277,-178.555,6.777,148.827
C00675=1158.034,151.438,-57.256,-178.557,6.775,148.827
C00676=1158.039,151.188,-57.235,-178.560,6.773,148.828
C00677=1158.043,150.939,-57.214,-178.562,6.771,148.828
C00678=1158.048,150.690,-57.192,-178.565,6.770,148.828
C00679=1158.053,150.441,-57.171,-178.568,6.768,148.829
C00680=1158.057,150.192,-57.151,-178.570,6.766,148.829
C00681=1158.062,149.943,-57.129,-178.574,6.764,148.829
C00682=1158.067,149.694,-57.108,-178.576,6.762,148.830
C00683=1158.071,149.444,-57.087,-178.579,6.760,148.830
C00684=1158.076,149.196,-57.066,-178.582,6.758,148.830
C00685=1158.081,148.946,-57.045,-178.584,6.757,148.831
C00686=1158.086,148.697,-57.024,-178.587,6.755,148.831
C00687=1158.090,148.449,-57.003,-178.590,6.753,148.832
C00688=1158.095,148.200,-56.982,-178.593,6.751,148.832
C00689=1158.100,147.951,-56.961,-178.595,6.750,148.832
C00690=1158.105,147.701,-56.940,-178.598,6.748,148.833
C00691=1158.109,147.452,-56.920,-178.601,6.745,148.833
C00692=1158.114,147.203,-56.898,-178.604,6.744,148.833
C00693=1158.118,146.954,-56.878,-178.607,6.742,148.834
C00694=1158.123,146.705,-56.857,-178.609,6.740,148.834
C00695=1158.128,146.456,-56.836,-178.612,6.739,148.835
C00696=1158.133,146.207,-56.815,-178.615,6.737,148.835
C00697=1158.137,145.958,-56.794,-178.618,6.735,148.835
C00698=1158.142,145.709,-56.773,-178.620,6.733,148.836
C00699=1158.148,145.460,-56.752,-178.623,6.732,148.836
C00700=1158.151,145.210,-56.732,-178.626,6.730,148.837
C00701=1158.157,144.961,-56.711,-178.628,6.728,148.837
C00702=1158.161,144.712,-56.690,-178.631,6.726,148.837
C00703=1158.166,144.463,-56.669,-178.634,6.725,148.838
C00704=1158.171,144.214,-56.649,-178.636,6.723,148.838
C00705=1158.175,143.965,-56.628,-178.640,6.720,148.838
C00706=1158.180,143.715,-56.608,-178.642,6.719,148.839
C00707=1158.185,143.467,-56.587,-178.645,6.717,148.839
C00708=1158.190,143.217,-56.566,-178.648,6.715,148.840
C00709=1158.194,142.968,-56.546,-178.651,6.713,148.840
C00710=1158.199,142.719,-56.525,-178.653,6.712,148.840
C00711=1158.204,142.470,-56.504,-178.656,6.710,148.841
C00712=1158.208,142.221,-56.484,-178.659,6.708,148.841
C00713=1158.214,141.972,-56.463,-178.661,6.707,148.842
C00714=1158.218,141.723,-56.443,-178.664,6.705,148.842
C00715=1158.223,141.474,-56.422,-178.667,6.703,148.842
C00716=1158.228,141.225,-56.401,-178.669,6.701,148.843
C00717=1158.232,140.976,-56.381,-178.672,6.700,148.843
C00718=1158.237,140.727,-56.360,-178.675,6.698,148.843
C00719=1158.242,140.478,-56.340,-178.678,6.696,148.844
C00720=1158.247,140.228,-56.319,-178.680,6.695,148.844
C00721=1158.251,139.979,-56.298,-178.683,6.693,148.845
C00722=1158.256,139.730,-56.278,-178.686,6.691,148.845
C00723=1158.261,139.481,-56.258,-178.688,6.689,148.845
C00724=1158.266,139.232,-56.237,-178.691,6.688,148.846
C00725=1158.270,138.983,-56.217,-178.694,6.686,148.846
C00726=1158.275,138.733,-56.196,-178.697,6.684,148.847
C00727=1158.280,138.484,-56.176,-178.699,6.682,148.847
C00728=1158.284,138.236,-56.155,-178.702,6.681,148.847
C00729=1158.289,137.986,-56.136,-178.705,6.679,148.848
C00730=1158.294,137.737,-56.115,-178.707,6.677,148.848
C00731=1158.298,137.488,-56.094,-178.710,6.676,148.849
C00732=1158.303,137.239,-56.074,-178.713,6.674,148.849
C00733=1158.308,136.990,-56.055,-178.716,6.672,148.849
C00734=1158.313,136.741,-56.034,-178.718,6.670,148.850
C00735=1158.318,136.492,-56.013,-178.721,6.669,148.850
C00736=1158.322,136.243,-55.993,-178.724,6.667,148.851
C00737=1158.327,135.993,-55.973,-178.727,6.666,148.851
C00738=1158.332,135.744,-55.952,-178.730,6.664,148.852
C00739=1158.337,135.495,-55.932,-178.732,6.662,148.852
C00740=1158.341,135.245,-55.912,-178.735,6.660,148.852
C00741=1158.346,134.996,-55.892,-178.738,6.659,148.853
C00742=1158.352,134.748,-55.871,-178.740,6.657,148.853
C00743=1158.356,134.498,-55.852,-178.743,6.655,148.853
C00744=1158.361,134.249,-55.831,-178.746,6.653,148.854
C00745=1158.366,134.000,-55.812,-178.748,6.652,148.854
C00746=1158.370,133.751,-55.791,-178.751,6.650,148.855
C00747=1158.374,133.502,-55.771,-178.754,6.648,148.855
C00748=1158.380,133.252,-55.751,-178.757,6.647,148.855
C00749=1158.385,133.004,-55.731,-178.759,6.645,148.856
C00750=1158.390,132.754,-55.711,-178.762,6.643,148.856
C00751=1158.394,132.505,-55.691,-178.765,6.641,148.857
C00752=1158.399,132.237,-55.670,-178.768,6.640,148.857
C00753=1158.404,131.968,-55.647,-178.771,6.638,148.858
C00754=1158.409,131.700,-55.626,-178.774,6.636,148.858
C00755=1158.415,131.431,-55.604,-178.777,6.634,148.858
C00756=1158.419,131.182,-55.584,-178.779,6.632,148.859
C00757=1158.424,130.932,-55.564,-178.783,6.631,148.859
C00758=1158.429,130.684,-55.544,-178.785,6.629,148.860
C00759=1158.434,130.434,-55.525,-178.788,6.628,148.860
C00760=1158.438,130.185,-55.504,-178.791,6.626,148.861
C00761=1158.443,129.936,-55.485,-178.793,6.624,148.861
C00762=1158.448,129.687,-55.465,-178.796,6.622,148.861
C00763=1158.453,129.438,-55.445,-178.799,6.621,148.862
C00764=1158.458,129.188,-55.425,-178.802,6.619,148.862
C00765=1158.462,128.940,-55.405,-178.804,6.617,148.863
C00766=1158.467,128.691,-55.386,-178.807,6.616,148.863
C00767=1158.472,128.441,-55.366,-178.810,6.614,148.863
C00768=1158.477,128.192,-55.346,-178.813,6.612,148.864
C00769=1158.481,127.943,-55.326,-178.815,6.612,148.864
C00770=1158.487,127.694,-55.307,-178.818,6.610,148.865
C00771=1158.491,127.445,-55.286,-178.820,6.608,148.865
C00772=1158.496,127.195,-55.267,-178.823,6.606,148.866
C00773=1158.501,126.946,-55.247,-178.826,6.605,148.866
C00774=1158.506,126.697,-55.227,-178.829,6.603,148.866
C00775=1158.510,126.448,-55.207,-178.831,6.601,148.867
C00776=1158.515,126.198,-55.188,-178.834,6.600,148.867
C00777=1158.520,125.949,-55.168,-178.837,6.598,148.868
C00778=1158.525,125.700,-55.148,-178.840,6.596,148.868
C00779=1158.530,125.451,-55.128,-178.843,6.595,148.869
C00780=1158.534,125.201,-55.109,-178.845,6.593,148.869
C00781=1158.540,124.952,-55.089,-178.848,6.591,148.869
C00782=1158.543,124.704,-55.070,-178.851,6.590,148.870
C00783=1158.548,124.454,-55.050,-178.853,6.589,148.870
C00784=1158.553,124.205,-55.031,-178.856,6.587,148.871
C00785=1158.558,123.956,-55.011,-178.859,6.586,148.871
C00786=1158.563,123.706,-54.991,-178.861,6.584,148.872
C00787=1158.568,123.457,-54.972,-178.864,6.582,148.872
C00788=1158.573,123.208,-54.952,-178.867,6.580,148.872
C00789=1158.577,122.959,-54.933,-178.870,6.579,148.873
C00790=1158.582,122.710,-54.913,-178.872,6.577,148.873
C00791=1158.587,122.461,-54.894,-178.875,6.575,148.874
C00792=1158.592,122.211,-54.874,-178.878,6.574,148.874
C00793=1158.597,121.962,-54.855,-178.881,6.572,148.875
C00794=1158.602,121.713,-54.835,-178.883,6.571,148.875
C00795=1158.606,121.464,-54.816,-178.886,6.570,148.875
C00796=1158.611,121.215,-54.797,-178.889,6.568,148.876
C00797=1158.616,120.965,-54.777,-178.891,6.566,148.876
C00798=1158.621,120.716,-54.758,-178.894,6.565,148.877
C00799=1158.625,120.467,-54.739,-178.897,6.563,148.877
C00800=1158.630,120.218,-54.719,-178.900,6.561,148.878
C00801=1158.635,119.968,-54.700,-178.903,6.560,148.878
C00802=1158.640,119.719,-54.680,-178.905,6.558,148.878
C00803=1158.645,119.470,-54.661,-178.907,6.557,148.879
C00804=1158.649,119.221,-54.642,-178.910,6.555,148.879
C00805=1158.655,118.972,-54.622,-178.913,6.554,148.880
C00806=1158.659,118.722,-54.603,-178.916,6.552,148.880
C00807=1158.664,118.474,-54.584,-178.919,6.551,148.881
C00808=1158.669,118.224,-54.564,-178.922,6.549,148.881
C00809=1158.673,117.975,-54.545,-178.924,6.547,148.881
C00810=1158.678,117.726,-54.526,-178.927,6.546,148.882
C00811=1158.683,117.476,-54.506,-178.929,6.545,148.882
C00812=1158.688,117.228,-54.487,-178.932,6.543,148.883
C00813=1158.692,116.978,-54.468,-178.935,6.542,148.883
C00814=1158.698,116.729,-54.450,-178.938,6.540,148.884
C00815=1158.703,116.479,-54.430,-178.940,6.538,148.884
C00816=1158.707,116.231,-54.411,-178.943,6.536,148.885
C00817=1158.712,115.981,-54.392,-178.946,6.535,148.885
C00818=1158.717,115.732,-54.372,-178.948,6.534,148.886
C00819=1158.721,115.483,-54.353,-178.951,6.532,148.886
C00820=1158.727,115.234,-54.335,-178.954,6.531,148.886
C00821=1158.732,114.984,-54.315,-178.957,6.529,148.887
C00822=1158.736,114.735,-54.296,-178.959,6.527,148.887
C00823=1158.741,114.486,-54.277,-178.962,6.526,148.888
C00824=1158.746,114.237,-54.259,-178.965,6.525,148.888
C00825=1158.751,113.987,-54.239,-178.967,6.523,148.889
C00826=1158.755,113.739,-54.220,-178.970,6.522,148.889
C00827=1158.760,113.489,-54.201,-178.973,6.520,148.889
C00828=1158.766,113.240,-54.182,-178.976,6.518,148.890
C00829=1158.770,112.990,-54.163,-178.979,6.517,148.890
C00830=1158.775,112.741,-54.144,-178.981,6.515,148.891
C00831=1158.780,112.492,-54.126,-178.984,6.514,148.891
C00832=1158.785,112.243,-54.106,-178.986,6.513,148.892
C00833=1158.789,111.994,-54.087,-178.989,6.511,148.892
C00834=1158.794,111.744,-54.068,-178.992,6.510,148.893
C00835=1158.799,111.495,-54.050,-178.995,6.508,148.893
C00836=1158.804,111.246,-54.030,-178.997,6.507,148.894
C00837=1158.809,110.997,-54.012,-179.000,6.505,148.894
C00838=1158.814,110.748,-53.993,-179.003,6.504,148.894
C00839=1158.818,110.498,-53.974,-179.006,6.502,148.895
C00840=1158.824,110.249,-53.955,-179.008,6.500,148.895
C00841=1158.828,110.000,-53.936,-179.011,6.499,148.896
C00842=1158.833,109.750,-53.918,-179.013,6.498,148.896
C00843=1158.838,109.502,-53.899,-179.016,6.496,148.897
C00844=1158.843,109.251,-53.880,-179.019,6.495,148.897
C00845=1158.847,109.003,-53.861,-179.022,6.493,148.898
C00846=1158.852,108.753,-53.843,-179.025,6.491,148.898
C00847=1158.857,108.504,-53.824,-179.027,6.491,148.898
C00848=1158.862,108.255,-53.806,-179.030,6.489,148.899
C00849=1158.867,108.005,-53.786,-179.033,6.487,148.900
C00850=1158.872,107.756,-53.768,-179.035,6.486,148.900
C00851=1158.876,107.508,-53.749,-179.038,6.484,148.900
C00852=1158.881,107.258,-53.730,-179.040,6.483,148.901
C00853=1158.886,107.009,-53.712,-179.044,6.482,148.901
C00854=1158.892,106.759,-53.693,-179.046,6.480,148.902
C00855=1158.896,106.510,-53.674,-179.049,6.478,148.902
C00856=1158.901,106.242,-53.655,-179.052,6.477,148.903
C00857=1158.907,105.973,-53.635,-179.055,6.475,148.903
C00858=1158.911,105.706,-53.614,-179.058,6.474,148.904
C00859=1158.917,105.437,-53.594,-179.061,6.472,148.904
C00860=1158.921,105.187,-53.576,-179.063,6.471,148.905
C00861=1158.927,104.938,-53.557,-179.066,6.470,148.905
C00862=1158.931,104.689,-53.538,-179.068,6.468,148.906
C00863=1158.936,104.439,-53.520,-179.072,6.467,148.906
C00864=1158.941,104.191,-53.502,-179.074,6.465,148.907
C00865=1158.946,103.941,-53.483,-179.076,6.464,148.907
C00866=1158.951,103.691,-53.465,-179.079,6.462,148.907
C00867=1158.955,103.442,-53.447,-179.082,6.461,148.908
C00868=1158.961,103.193,-53.428,-179.085,6.459,148.908
C00869=1158.965,102.944,-53.409,-179.087,6.458,148.909
C00870=1158.970,102.694,-53.391,-179.090,6.457,148.909
C00871=1158.975,102.446,-53.373,-179.093,6.455,148.910
C00872=1158.980,102.196,-53.354,-179.096,6.454,148.910
C00873=1158.985,101.946,-53.336,-179.098,6.453,148.911
C00874=1158.990,101.697,-53.318,-179.101,6.451,148.911
C00875=1158.994,101.448,-53.300,-179.104,6.450,148.912
C00876=1158.999,101.200,-53.281,-179.107,6.448,148.912
C00877=1159.004,100.949,-53.262,-179.109,6.447,148.913
C00878=1159.009,100.700,-53.244,-179.112,6.445,148.913
C00879=1159.014,100.451,-53.226,-179.115,6.444,148.914
C00880=1159.019,100.202,-53.208,-179.117,6.442,148.914
C00881=1159.023,99.953,-53.189,-179.120,6.442,148.915
C00882=1159.028,99.703,-53.170,-179.122,6.440,148.915
C00883=1159.033,99.454,-53.152,-179.126,6.439,148.916
C00884=1159.038,99.205,-53.135,-179.128,6.437,148.916
C00885=1159.043,98.956,-53.117,-179.130,6.436,148.916
C00886=1159.048,98.706,-53.099,-179.134,6.435,148.917
C00887=1159.052,98.457,-53.080,-179.136,6.433,148.917
C00888=1159.057,98.207,-53.062,-179.139,6.431,148.918
C00889=1159.063,97.958,-53.044,-179.141,6.430,148.918
C00890=1159.068,97.709,-53.026,-179.144,6.429,148.919
C00891=1159.073,97.460,-53.007,-179.147,6.427,148.919
C00892=1159.077,97.211,-52.989,-179.149,6.426,148.920
C00893=1159.082,96.961,-52.971,-179.152,6.425,148.920
C00894=1159.087,96.712,-52.953,-179.155,6.423,148.921
C00895=1159.092,96.463,-52.935,-179.158,6.422,148.921
C00896=1159.096,96.214,-52.917,-179.160,6.421,148.922
C00897=1159.101,95.964,-52.899,-179.163,6.419,148.922
C00898=1159.106,95.715,-52.881,-179.166,6.418,148.923
C00899=1159.111,95.466,-52.863,-179.168,6.417,148.923
C00900=1159.116,95.216,-52.845,-179.171,6.415,148.924
C00901=1159.121,94.966,-52.827,-179.174,6.414,148.924
C00902=1159.126,94.717,-52.809,-179.177,6.412,148.925
C00903=1159.131,94.468,-52.791,-179.179,6.411,148.925
C00904=1159.135,94.219,-52.773,-179.182,6.410,148.926
C00905=1159.140,93.970,-52.755,-179.185,6.408,148.926
C00906=1159.145,93.720,-52.737,-179.187,6.407,148.927
C00907=1159.150,93.471,-52.719,-179.190,6.406,148.927
C00908=1159.155,93.222,-52.701,-179.193,6.404,148.928
C00909=1159.160,92.973,-52.683,-179.195,6.403,148.928
C00910=1159.165,92.722,-52.666,-179.198,6.402,148.928
C00911=1159.170,92.473,-52.648,-179.201,6.400,148.929
C00912=1159.174,92.224,-52.630,-179.204,6.399,148.929
C00913=1159.179,91.975,-52.612,-179.206,6.398,148.930
C00914=1159.184,91.726,-52.594,-179.209,6.397,148.931
C00915=1159.189,91.477,-52.576,-179.212,6.395,148.931
C00916=1159.194,91.227,-52.559,-179.214,6.394,148.931
C00917=1159.199,90.978,-52.541,-179.217,6.392,148.932
C00918=1159.204,90.728,-52.523,-179.220,6.391,148.932
C00919=1159.209,90.479,-52.505,-179.222,6.390,148.933
C00920=1159.214,90.229,-52.487,-179.225,6.388,148.933
C00921=1159.219,89.980,-52.469,-179.228,6.387,148.934
C00922=1159.223,89.731,-52.452,-179.230,6.386,148.934
C00923=1159.228,89.482,-52.434,-179.233,6.384,148.935
C00924=1159.234,89.232,-52.417,-179.236,6.383,148.935
C00925=1159.239,88.983,-52.399,-179.238,6.382,148.936
C00926=1159.243,88.734,-52.381,-179.241,6.381,148.936
C00927=1159.249,88.484,-52.363,-179.244,6.379,148.937
C00928=1159.254,88.235,-52.346,-179.246,6.378,148.937
C00929=1159.258,87.986,-52.328,-179.249,6.377,148.938
C00930=1159.263,87.736,-52.311,-179.252,6.375,148.938
C00931=1159.268,87.487,-52.293,-179.254,6.374,148.939
C00932=1159.273,87.238,-52.275,-179.257,6.373,148.939
C00933=1159.278,86.988,-52.258,-179.260,6.371,148.940
C00934=1159.282,86.739,-52.240,-179.262,6.371,148.940
C00935=1159.287,86.490,-52.222,-179.265,6.369,148.941
C00936=1159.292,86.240,-52.205,-179.268,6.368,148.941
C00937=1159.297,85.991,-52.187,-179.271,6.367,148.942
C00938=1159.302,85.742,-52.170,-179.273,6.365,148.942
C00939=1159.307,85.493,-52.152,-179.276,6.364,148.943
C00940=1159.312,85.243,-52.135,-179.279,6.363,148.943
C00941=1159.317,84.994,-52.117,-179.281,6.361,148.944
C00942=1159.322,84.744,-52.100,-179.284,6.361,148.944
C00943=1159.326,84.495,-52.082,-179.287,6.359,148.945
C00944=1159.331,84.245,-52.065,-179.289,6.357,148.945
C00945=1159.336,83.996,-52.047,-179.292,6.357,148.946
C00946=1159.341,83.747,-52.031,-179.295,6.355,148.946
C00947=1159.346,83.498,-52.013,-179.297,6.354,148.947
C00948=1159.351,83.248,-51.996,-179.300,6.353,148.947
C00949=1159.356,82.999,-51.978,-179.303,6.351,148.948
C00950=1159.361,82.750,-51.961,-179.305,6.350,148.948
C00951=1159.366,82.500,-51.943,-179.308,6.349,148.949
C00952=1159.371,82.251,-51.926,-179.311,6.347,148.949
C00953=1159.375,82.002,-51.908,-179.313,6.346,148.950
C00954=1159.380,81.752,-51.891,-179.316,6.345,148.950
C00955=1159.386,81.503,-51.874,-179.319,6.344,148.951
C00956=1159.390,81.254,-51.857,-179.321,6.342,148.951
C00957=1159.396,81.004,-51.840,-179.324,6.341,148.952
C00958=1159.400,80.755,-51.822,-179.327,6.340,148.952
C00959=1159.405,80.506,-51.805,-179.329,6.339,148.953
C00960=1159.410,80.237,-51.786,-179.333,6.337,148.953
C00961=1159.416,79.969,-51.768,-179.335,6.336,148.954
C00962=1159.421,79.701,-51.749,-179.338,6.335,148.954
C00963=1159.426,79.432,-51.730,-179.341,6.334,148.955
C00964=1159.432,79.183,-51.714,-179.344,6.332,148.956
C00965=1159.436,78.933,-51.697,-179.346,6.331,148.956
C00966=1159.441,78.684,-51.679,-179.349,6.330,148.957
C00967=1159.446,78.435,-51.662,-179.351,6.329,148.957
C00968=1159.451,78.185,-51.645,-179.354,6.327,148.957
C00969=1159.456,77.936,-51.629,-179.357,6.326,148.958
C00970=1159.461,77.687,-51.611,-179.359,6.325,148.959
C00971=1159.465,77.437,-51.594,-179.362,6.323,148.959
C00972=1159.471,77.187,-51.577,-179.365,6.323,148.960
C00973=1159.476,76.938,-51.559,-179.368,6.321,148.960
C00974=1159.481,76.690,-51.542,-179.370,6.321,148.961
C00975=1159.486,76.440,-51.525,-179.373,6.319,148.961
C00976=1159.490,76.190,-51.509,-179.376,6.317,148.962
C00977=1159.496,75.940,-51.491,-179.378,6.317,148.962
C00978=1159.500,75.691,-51.475,-179.381,6.315,148.963
C00979=1159.506,75.442,-51.458,-179.383,6.314,148.963
C00980=1159.510,75.193,-51.440,-179.386,6.313,148.964
C00981=1159.515,74.944,-51.424,-179.389,6.312,148.964
C00982=1159.520,74.694,-51.406,-179.392,6.311,148.965
C00983=1159.525,74.445,-51.390,-179.395,6.309,148.965
C00984=1159.530,74.195,-51.373,-179.397,6.308,148.966
C00985=1159.535,73.946,-51.356,-179.400,6.307,148.966
C00986=1159.540,73.696,-51.339,-179.402,6.306,148.967
C00987=1159.545,73.447,-51.323,-179.405,6.304,148.967
C00988=1159.550,73.197,-51.305,-179.407,6.304,148.968
C00989=1159.554,72.948,-51.288,-179.410,6.302,148.968
C00990=1159.559,72.700,-51.272,-179.413,6.302,148.969
C00991=1159.565,72.450,-51.254,-179.416,6.300,148.969
C00992=1159.569,72.200,-51.238,-179.418,6.298,148.970
C00993=1159.574,71.951,-51.220,-179.421,6.298,148.970
C00994=1159.579,71.702,-51.204,-179.424,6.296,148.971
C00995=1159.584,71.452,-51.187,-179.426,6.296,148.972
C00996=1159.589,71.202,-51.170,-179.429,6.294,148.972
C00997=1159.594,70.954,-51.154,-179.431,6.293,148.972
C00998=1159.599,70.704,-51.137,-179.434,6.292,148.973
C00999=1159.604,70.454,-51.120,-179.436,6.291,148.974
C01000=1159.609,70.206,-51.104,-179.439,6.289,148.974
C01001=1159.614,69.955,-51.087,-179.442,6.289,148.975
C01002=1159.619,69.706,-51.070,-179.445,6.287,148.975
C01003=1159.624,69.457,-51.054,-179.447,6.287,148.976
C01004=1159.629,69.207,-51.037,-179.450,6.285,148.976
C01005=1159.634,68.958,-51.020,-179.453,6.283,148.977
C01006=1159.639,68.709,-51.004,-179.455,6.283,148.977
C01007=1159.643,68.459,-50.987,-179.458,6.281,148.978
C01008=1159.648,68.210,-50.970,-179.461,6.280,148.978
C01009=1159.654,67.961,-50.954,-179.463,6.279,148.979
C01010=1159.658,67.711,-50.938,-179.466,6.278,148.979
C01011=1159.664,67.462,-50.921,-179.469,6.277,148.980
C01012=1159.669,67.212,-50.904,-179.471,6.276,148.980
C01013=1159.673,66.963,-50.887,-179.474,6.274,148.981
C01014=1159.678,66.714,-50.871,-179.476,6.274,148.981
C01015=1159.683,66.464,-50.854,-179.480,6.272,148.982
C01016=1159.688,66.214,-50.838,-179.482,6.271,148.982
C01017=1159.693,65.965,-50.822,-179.484,6.270,148.983
C01018=1159.698,65.716,-50.805,-179.487,6.269,148.984
C01019=1159.703,65.467,-50.789,-179.490,6.268,148.984
C01020=1159.708,65.217,-50.771,-179.492,6.267,148.985
C01021=1159.713,64.967,-50.755,-179.495,6.265,148.985
C01022=1159.718,64.718,-50.739,-179.497,6.265,148.986
C01023=1159.722,64.469,-50.722,-179.501,6.263,148.986
C01024=1159.728,64.219,-50.707,-179.503,6.262,148.987
C01025=1159.733,63.970,-50.690,-179.506,6.261,148.987
C01026=1159.738,63.721,-50.673,-179.508,6.260,148.988
C01027=1159.743,63.471,-50.657,-179.511,6.259,148.988
C01028=1159.748,63.222,-50.641,-179.513,6.258,148.989
C01029=1159.752,62.972,-50.624,-179.516,6.256,148.989
C01030=1159.757,62.723,-50.608,-179.519,6.256,148.990
C01031=1159.762,62.474,-50.592,-179.522,6.254,148.990
C01032=1159.767,62.224,-50.575,-179.524,6.254,148.991
C01033=1159.773,61.974,-50.559,-179.527,6.252,148.991
C01034=1159.777,61.725,-50.543,-179.529,6.251,148.992
C01035=1159.782,61.476,-50.526,-179.532,6.250,148.993
C01036=1159.787,61.226,-50.510,-179.535,6.249,148.993
C01037=1159.792,60.977,-50.494,-179.537,6.248,148.994
C01038=1159.797,60.728,-50.477,-179.540,6.247,148.994
C01039=1159.802,60.478,-50.462,-179.543,6.246,148.995
C01040=1159.807,60.229,-50.445,-179.545,6.245,148.995
C01041=1159.812,59.979,-50.430,-179.547,6.244,148.996
C01042=1159.817,59.730,-50.413,-179.551,6.242,148.996
C01043=1159.823,59.480,-50.397,-179.553,6.242,148.997
C01044=1159.827,59.231,-50.380,-179.556,6.240,148.997
C01045=1159.833,58.981,-50.364,-179.558,6.239,148.998
C01046=1159.837,58.732,-50.348,-179.561,6.238,148.998
C01047=1159.842,58.482,-50.332,-179.564,6.237,148.999
C01048=1159.847,58.233,-50.315,-179.567,6.236,149.000
C01049=1159.852,57.984,-50.300,-179.569,6.235,149.000
C01050=1159.857,57.735,-50.284,-179.571,6.234,149.000
C01051=1159.862,57.485,-50.268,-179.574,6.233,149.001
C01052=1159.867,57.236,-50.251,-179.576,6.232,149.002
C01053=1159.872,56.986,-50.235,-179.580,6.231,149.002
C01054=1159.877,56.737,-50.219,-179.582,6.230,149.003
C01055=1159.882,56.487,-50.203,-179.585,6.229,149.003
C01056=1159.887,56.237,-50.188,-179.587,6.228,149.004
C01057=1159.892,55.989,-50.171,-179.590,6.226,149.004
C01058=1159.897,55.739,-50.155,-179.593,6.226,149.005
C01059=1159.902,55.490,-50.139,-179.595,6.225,149.005
C01060=1159.906,55.240,-50.124,-179.598,6.223,149.006
C01061=1159.912,54.991,-50.108,-179.600,6.223,149.006
C01062=1159.917,54.742,-50.092,-179.603,6.221,149.007
C01063=1159.921,54.492,-50.076,-179.606,6.220,149.008
C01064=1159.927,54.223,-50.059,-179.609,6.219,149.008
C01065=1159.933,53.955,-50.042,-179.611,6.218,149.009
C01066=1159.938,53.686,-50.024,-179.614,6.217,149.009
C01067=1159.943,53.417,-50.007,-179.617,6.216,149.010
C01068=1159.948,53.168,-49.991,-179.620,6.215,149.010
C01069=1159.954,52.919,-49.975,-179.622,6.214,149.011
C01070=1159.958,52.669,-49.959,-179.625,6.213,149.011
C01071=1159.964,52.419,-49.944,-179.628,6.212,149.012
C01072=1159.968,52.170,-49.927,-179.630,6.211,149.013
C01073=1159.973,51.921,-49.912,-179.632,6.210,149.013
C01074=1159.978,51.671,-49.897,-179.636,6.208,149.014
C01075=1159.983,51.421,-49.881,-179.638,6.207,149.014
C01076=1159.988,51.173,-49.864,-179.640,6.207,149.015
C01077=1159.994,50.923,-49.849,-179.643,6.205,149.015
C01078=1159.998,50.673,-49.833,-179.646,6.205,149.016
C01079=1160.003,50.424,-49.818,-179.649,6.203,149.016
C01080=1160.008,50.175,-49.802,-179.651,6.203,149.017
C01081=1160.013,49.925,-49.786,-179.653,6.202,149.017
C01082=1160.018,49.676,-49.770,-179.657,6.201,149.018
C01083=1160.024,49.426,-49.754,-179.659,6.200,149.019
C01084=1160.028,49.176,-49.739,-179.662,6.198,149.019
C01085=1160.033,48.927,-49.723,-179.664,6.198,149.020
C01086=1160.038,48.678,-49.708,-179.666,6.197,149.020
C01087=1160.044,48.428,-49.692,-179.670,6.195,149.021
C01088=1160.048,48.178,-49.677,-179.672,6.195,149.021
C01089=1160.053,47.930,-49.661,-179.674,6.194,149.022
C01090=1160.058,47.680,-49.645,-179.677,6.192,149.022
C01091=1160.063,47.430,-49.629,-179.680,6.192,149.023
C01092=1160.068,47.181,-49.614,-179.682,6.190,149.023
C01093=1160.073,46.932,-49.599,-179.685,6.190,149.024
C01094=1160.079,46.682,-49.583,-179.687,6.189,149.025
C01095=1160.083,46.433,-49.568,-179.691,6.188,149.025
C01096=1160.088,46.183,-49.552,-179.693,6.187,149.026
C01097=1160.093,45.934,-49.536,-179.696,6.185,149.026
C01098=1160.099,45.684,-49.521,-179.698,6.185,149.027
C01099=1160.103,45.435,-49.505,-179.701,6.184,149.028
C01100=1160.108,45.185,-49.490,-179.703,6.182,149.028
C01101=1160.114,44.936,-49.474,-179.706,6.182,149.029
C01102=1160.118,44.687,-49.459,-179.708,6.181,149.029
C01103=1160.123,44.437,-49.443,-179.711,6.180,149.030
C01104=1160.128,44.187,-49.428,-179.714,6.179,149.030
C01105=1160.133,43.938,-49.413,-179.716,6.178,149.031
C01106=1160.138,43.689,-49.397,-179.719,6.177,149.031
C01107=1160.144,43.439,-49.382,-179.721,6.176,149.032
C01108=1160.148,43.189,-49.366,-179.724,6.175,149.032
C01109=1160.153,42.940,-49.351,-179.727,6.174,149.033
C01110=1160.158,42.691,-49.336,-179.729,6.173,149.034
C01111=1160.164,42.441,-49.321,-179.732,6.172,149.034
C01112=1160.169,42.192,-49.305,-179.735,6.171,149.035
C01113=1160.174,41.942,-49.290,-179.737,6.170,149.035
C01114=1160.178,41.692,-49.274,-179.740,6.169,149.036
C01115=1160.183,41.443,-49.259,-179.742,6.168,149.036
C01116=1160.188,41.194,-49.244,-179.745,6.168,149.037
C01117=1160.194,40.944,-49.228,-179.748,6.166,149.037
C01118=1160.199,40.695,-49.214,-179.750,6.166,149.038
C01119=1160.204,40.445,-49.198,-179.752,6.165,149.038
C01120=1160.208,40.196,-49.183,-179.756,6.163,149.039
C01121=1160.214,39.946,-49.167,-179.758,6.163,149.040
C01122=1160.218,39.697,-49.152,-179.760,6.162,149.040
C01123=1160.224,39.447,-49.137,-179.763,6.161,149.041
C01124=1160.229,39.198,-49.122,-179.766,6.160,149.041
C01125=1160.234,38.949,-49.107,-179.768,6.159,149.042
C01126=1160.239,38.699,-49.092,-179.771,6.158,149.042
C01127=1160.244,38.449,-49.077,-179.773,6.157,149.043
C01128=1160.248,38.200,-49.062,-179.776,6.157,149.044
C01129=1160.254,37.950,-49.046,-179.779,6.155,149.044
C01130=1160.258,37.701,-49.031,-179.781,6.154,149.045
C01131=1160.264,37.451,-49.016,-179.784,6.154,149.045
C01132=1160.269,37.202,-49.001,-179.787,6.152,149.046
C01133=1160.274,36.953,-48.986,-179.789,6.151,149.046
C01134=1160.279,36.703,-48.971,-179.792,6.151,149.047
C01135=1160.284,36.453,-48.956,-179.794,6.149,149.047
C01136=1160.289,36.204,-48.941,-179.797,6.149,149.048
C01137=1160.295,35.954,-48.926,-179.799,6.148,149.049
C01138=1160.299,35.705,-48.911,-179.802,6.148,149.049
C01139=1160.304,35.455,-48.895,-179.805,6.146,149.050
C01140=1160.309,35.205,-48.881,-179.807,6.145,149.050
C01141=1160.314,34.956,-48.866,-179.809,6.145,149.051
C01142=1160.319,34.707,-48.850,-179.813,6.143,149.051
C01143=1160.324,34.457,-48.836,-179.815,6.142,149.052
C01144=1160.330,34.208,-48.820,-179.817,6.142,149.053
C01145=1160.335,33.958,-48.806,-179.820,6.140,149.053
C01146=1160.339,33.709,-48.791,-179.823,6.140,149.054
C01147=1160.345,33.459,-48.776,-179.825,6.139,149.054
C01148=1160.350,33.210,-48.761,-179.828,6.138,149.055
C01149=1160.355,32.961,-48.745,-179.830,6.137,149.055
C01150=1160.360,32.711,-48.731,-179.833,6.136,149.056
C01151=1160.365,32.462,-48.716,-179.835,6.136,149.056
C01152=1160.370,32.212,-48.701,-179.838,6.134,149.057
C01153=1160.375,31.963,-48.686,-179.841,6.133,149.058
C01154=1160.380,31.713,-48.672,-179.843,6.133,149.058
C01155=1160.385,31.464,-48.656,-179.845,6.132,149.059
C01156=1160.390,31.214,-48.642,-179.849,6.131,149.059
C01157=1160.395,30.965,-48.627,-179.851,6.130,149.060
C01158=1160.400,30.715,-48.612,-179.853,6.129,149.060
C01159=1160.405,30.466,-48.597,-179.856,6.128,149.061
C01160=1160.410,30.216,-48.583,-179.859,6.127,149.062
C01161=1160.415,29.966,-48.569,-179.861,6.127,149.062
C01162=1160.420,29.717,-48.553,-179.864,6.126,149.063
C01163=1160.425,29.467,-48.539,-179.866,6.124,149.063
C01164=1160.430,29.218,-48.524,-179.869,6.124,149.064
C01165=1160.436,28.968,-48.509,-179.871,6.123,149.064
C01166=1160.441,28.718,-48.495,-179.874,6.123,149.065
C01167=1160.445,28.469,-48.480,-179.877,6.121,149.065
C01168=1160.450,28.200,-48.464,-179.879,6.120,149.066
C01169=1160.456,27.931,-48.448,-179.882,6.119,149.067
C01170=1160.461,27.662,-48.432,-179.885,6.118,149.067
C01171=1160.467,27.394,-48.417,-179.887,6.118,149.068
C01172=1160.473,27.144,-48.402,-179.891,6.117,149.069
C01173=1160.478,26.895,-48.388,-179.893,6.116,149.069
C01174=1160.483,26.645,-48.373,-179.895,6.115,149.070
C01175=1160.487,26.396,-48.358,-179.897,6.114,149.070
C01176=1160.492,26.146,-48.344,-179.901,6.113,149.071
C01177=1160.498,25.896,-48.329,-179.903,6.112,149.071
C01178=1160.503,25.647,-48.314,-179.906,6.112,149.072
C01179=1160.508,25.397,-48.300,-179.908,6.111,149.072
C01180=1160.513,25.148,-48.286,-179.911,6.110,149.073
C01181=1160.518,24.898,-48.271,-179.913,6.109,149.074
C01182=1160.523,24.650,-48.257,-179.916,6.108,149.074
C01183=1160.529,24.399,-48.242,-179.918,6.108,149.075
C01184=1160.533,24.150,-48.228,-179.921,6.106,149.075
C01185=1160.538,23.900,-48.213,-179.923,6.106,149.076
C01186=1160.543,23.651,-48.198,-179.926,6.105,149.077
C01187=1160.548,23.401,-48.184,-179.929,6.105,149.077
C01188=1160.553,23.152,-48.170,-179.931,6.104,149.078
C01189=1160.558,22.902,-48.155,-179.934,6.102,149.078
C01190=1160.564,22.653,-48.141,-179.936,6.102,149.079
C01191=1160.569,22.403,-48.127,-179.939,6.101,149.079
C01192=1160.574,22.154,-48.112,-179.941,6.100,149.080
C01193=1160.579,21.904,-48.097,-179.944,6.099,149.081
C01194=1160.584,21.654,-48.083,-179.946,6.098,149.081
C01195=1160.589,21.405,-48.069,-179.949,6.098,149.082
C01196=1160.594,21.156,-48.055,-179.951,6.097,149.082
C01197=1160.599,20.906,-48.041,-179.954,6.096,149.083
C01198=1160.604,20.656,-48.026,-179.957,6.095,149.083
C01199=1160.609,20.406,-48.012,-179.959,6.094,149.084
C01200=1160.614,20.157,-47.997,-179.961,6.094,149.084
C01201=1160.619,19.908,-47.983,-179.964,6.093,149.085
C01202=1160.624,19.659,-47.969,-179.967,6.091,149.086
C01203=1160.629,19.409,-47.955,-179.970,6.091,149.086
C01204=1160.634,19.159,-47.940,-179.972,6.090,149.087
C01205=1160.639,18.909,-47.926,-179.974,6.090,149.087
C01206=1160.644,18.660,-47.912,-179.977,6.089,149.088
C01207=1160.650,18.411,-47.898,-179.980,6.088,149.089
C01208=1160.655,18.161,-47.884,-179.982,6.087,149.089
C01209=1160.660,17.911,-47.869,-179.985,6.086,149.090
C01210=1160.665,17.662,-47.855,-179.987,6.086,149.090
C01211=1160.670,17.413,-47.841,-179.989,6.085,149.091
C01212=1160.675,17.163,-47.827,-179.993,6.084,149.092
C01213=1160.680,16.913,-47.813,-179.995,6.083,149.092
C01214=1160.685,16.663,-47.798,-179.997,6.082,149.093
C01215=1160.691,16.414,-47.784,-180.000,6.082,149.093
C01216=1160.695,16.165,-47.770,179.998,6.081,149.094
C01217=1160.700,15.915,-47.756,179.996,6.080,149.094
C01218=1160.705,15.665,-47.742,179.992,6.079,149.095
C01219=1160.711,15.416,-47.728,179.990,6.078,149.095
C01220=1160.716,15.166,-47.714,179.988,6.078,149.096
C01221=1160.721,14.916,-47.700,179.985,6.077,149.097
C01222=1160.726,14.667,-47.686,179.983,6.076,149.097
C01223=1160.731,14.418,-47.672,179.979,6.075,149.098
C01224=1160.736,14.168,-47.658,179.977,6.074,149.098
C01225=1160.741,13.918,-47.644,179.975,6.074,149.099
C01226=1160.746,13.669,-47.630,179.972,6.073,149.100
C01227=1160.751,13.420,-47.615,179.970,6.073,149.100
C01228=1160.757,13.169,-47.602,179.968,6.072,149.101
C01229=1160.762,12.920,-47.588,179.964,6.070,149.101
C01230=1160.767,12.671,-47.574,179.962,6.070,149.102
C01231=1160.771,12.421,-47.560,179.960,6.069,149.102
C01232=1160.776,12.172,-47.546,179.957,6.068,149.103
C01233=1160.782,11.923,-47.532,179.955,6.068,149.104
C01234=1160.787,11.672,-47.518,179.952,6.067,149.104
C01235=1160.792,11.423,-47.504,179.949,6.066,149.105
C01236=1160.798,11.174,-47.490,179.947,6.065,149.105
C01237=1160.802,10.924,-47.476,179.945,6.064,149.106
C01238=1160.807,10.674,-47.463,179.942,6.064,149.107
C01239=1160.813,10.425,-47.449,179.940,6.063,149.107
C01240=1160.818,10.175,-47.435,179.937,6.063,149.108
C01241=1160.823,9.925,-47.420,179.935,6.062,149.108
C01242=1160.828,9.676,-47.407,179.932,6.061,149.109
C01243=1160.833,9.426,-47.393,179.929,6.060,149.109
C01244=1160.838,9.177,-47.380,179.927,6.059,149.110
C01245=1160.843,8.928,-47.365,179.925,6.059,149.110
C01246=1160.848,8.677,-47.352,179.922,6.058,149.111
C01247=1160.853,8.429,-47.338,179.919,6.058,149.112
C01248=1160.858,8.179,-47.324,179.917,6.057,149.112
C01249=1160.863,7.929,-47.311,179.914,6.056,149.113
C01250=1160.869,7.680,-47.297,179.912,6.055,149.113
C01251=1160.873,7.430,-47.283,179.909,6.054,149.114
C01252=1160.879,7.181,-47.270,179.907,6.053,149.115
C01253=1160.884,6.931,-47.256,179.904,6.053,149.115
C01254=1160.889,6.681,-47.243,179.902,6.052,149.116
C01255=1160.894,6.432,-47.229,179.899,6.052,149.116
C01256=1160.899,6.182,-47.214,179.897,6.051,149.117
C01257=1160.905,5.932,-47.201,179.894,6.050,149.118
C01258=1160.909,5.683,-47.187,179.891,6.049,149.118
C01259=1160.914,5.433,-47.174,179.889,6.048,149.119
C01260=1160.920,5.184,-47.160,179.887,6.048,149.119
C01261=1160.924,4.934,-47.146,179.884,6.047,149.120
C01262=1160.930,4.685,-47.133,179.882,6.047,149.121
C01263=1160.935,4.435,-47.119,179.880,6.046,149.121
C01264=1160.940,4.186,-47.106,179.877,6.045,149.122
C01265=1160.945,3.936,-47.092,179.874,6.044,149.122
C01266=1160.951,3.686,-47.079,179.872,6.043,149.123
C01267=1160.955,3.437,-47.065,179.869,6.042,149.123
C01268=1160.960,3.187,-47.052,179.867,6.042,149.124
C01269=1160.965,2.938,-47.038,179.864,6.042,149.125
C01270=1160.970,2.688,-47.025,179.862,6.041,149.125
C01271=1160.976,2.439,-47.011,179.859,6.040,149.126
C01272=1160.981,2.169,-46.997,179.857,6.039,149.126
C01273=1160.986,1.899,-46.982,179.854,6.038,149.127
C01274=1160.993,1.631,-46.967,179.851,6.038,149.128
C01275=1160.998,1.361,-46.953,179.848,6.037,149.128
C01276=1161.002,1.111,-46.939,179.846,6.036,149.129
C01277=1161.008,0.862,-46.926,179.844,6.036,149.130
C01278=1161.013,0.612,-46.912,179.841,6.034,149.130
C01279=1161.018,0.363,-46.899,179.838,6.034,149.131
C01280=1161.024,0.112,-46.886,179.836,6.033,149.131
C01281=1161.028,-0.136,-46.873,179.833,6.033,149.132
C01282=1161.034,-0.387,-46.859,179.831,6.032,149.132
C01283=1161.039,-0.635,-46.846,179.829,6.031,149.133
C01284=1161.044,-0.885,-46.832,179.826,6.031,149.134
C01285=1161.049,-1.135,-46.820,179.824,6.030,149.134
C01286=1161.055,-1.384,-46.806,179.821,6.030,149.135
C01287=1161.059,-1.634,-46.793,179.819,6.029,149.135
C01288=1161.065,-1.884,-46.779,179.816,6.028,149.136
C01289=1161.069,-2.133,-46.766,179.814,6.028,149.136
C01290=1161.075,-2.383,-46.753,179.811,6.026,149.137
C01291=1161.079,-2.633,-46.740,179.809,6.025,149.138
C01292=1161.085,-2.882,-46.726,179.806,6.025,149.138
C01293=1161.090,-3.132,-46.713,179.803,6.025,149.139
C01294=1161.095,-3.381,-46.700,179.801,6.024,149.139
C01295=1161.101,-3.631,-46.687,179.799,6.023,149.140
C01296=1161.106,-3.880,-46.673,179.796,6.022,149.141
C01297=1161.111,-4.130,-46.660,179.794,6.022,149.141
C01298=1161.116,-4.380,-46.646,179.792,6.021,149.142
C01299=1161.121,-4.629,-46.634,179.789,6.021,149.142
C01300=1161.127,-4.878,-46.620,179.787,6.020,149.143
C01301=1161.131,-5.128,-46.607,179.784,6.020,149.144
C01302=1161.136,-5.378,-46.594,179.782,6.019,149.144
C01303=1161.141,-5.628,-46.581,179.779,6.018,149.145
C01304=1161.146,-5.877,-46.568,179.777,6.018,149.145
C01305=1161.152,-6.126,-46.554,179.774,6.017,149.146
C01306=1161.157,-6.376,-46.541,179.771,6.016,149.147
C01307=1161.163,-6.626,-46.528,179.769,6.015,149.147
C01308=1161.167,-6.876,-46.515,179.766,6.014,149.148
C01309=1161.172,-7.125,-46.503,179.764,6.014,149.148
C01310=1161.178,-7.374,-46.489,179.761,6.013,149.149
C01311=1161.182,-7.624,-46.476,179.759,6.012,149.149
C01312=1161.187,-7.874,-46.463,179.757,6.012,149.150
C01313=1161.193,-8.123,-46.450,179.754,6.012,149.151
C01314=1161.198,-8.373,-46.437,179.752,6.011,149.151
C01315=1161.203,-8.623,-46.424,179.749,6.010,149.152
C01316=1161.208,-8.873,-46.411,179.747,6.009,149.152
C01317=1161.213,-9.122,-46.398,179.744,6.009,149.153
C01318=1161.218,-9.372,-46.386,179.742,6.008,149.154
C01319=1161.224,-9.622,-46.372,179.739,6.008,149.154
C01320=1161.228,-9.871,-46.359,179.737,6.007,149.155
C01321=1161.234,-10.120,-46.346,179.735,6.006,149.155
C01322=1161.239,-10.370,-46.333,179.732,6.006,149.156
C01323=1161.244,-10.620,-46.320,179.730,6.005,149.157
C01324=1161.249,-10.869,-46.307,179.727,6.005,149.157
C01325=1161.254,-11.119,-46.294,179.725,6.004,149.158
C01326=1161.260,-11.369,-46.281,179.722,6.003,149.158
C01327=1161.265,-11.618,-46.269,179.720,6.003,149.159
C01328=1161.270,-11.867,-46.256,179.717,6.002,149.160
C01329=1161.275,-12.118,-46.242,179.715,6.001,149.160
C01330=1161.280,-12.367,-46.230,179.713,6.001,149.161
C01331=1161.285,-12.616,-46.217,179.710,6.000,149.161
C01332=1161.290,-12.866,-46.204,179.708,6.000,149.162
C01333=1161.296,-13.116,-46.191,179.705,5.999,149.163
C01334=1161.301,-13.365,-46.178,179.703,5.998,149.163
C01335=1161.306,-13.615,-46.166,179.700,5.998,149.164
C01336=1161.311,-13.865,-46.154,179.698,5.997,149.164
C01337=1161.317,-14.115,-46.140,179.695,5.997,149.165
C01338=1161.322,-14.364,-46.128,179.693,5.996,149.165
C01339=1161.326,-14.614,-46.115,179.691,5.996,149.166
C01340=1161.331,-14.863,-46.102,179.688,5.995,149.167
C01341=1161.336,-15.113,-46.090,179.686,5.994,149.167
C01342=1161.342,-15.362,-46.076,179.683,5.994,149.168
C01343=1161.347,-15.612,-46.063,179.681,5.993,149.168
C01344=1161.352,-15.862,-46.051,179.678,5.993,149.169
C01345=1161.357,-16.111,-46.038,179.676,5.992,149.170
C01346=1161.363,-16.361,-46.026,179.673,5.991,149.170
C01347=1161.368,-16.611,-46.013,179.671,5.991,149.171
C01348=1161.373,-16.861,-46.000,179.669,5.990,149.171
C01349=1161.378,-17.110,-45.988,179.666,5.989,149.172
C01350=1161.383,-17.359,-45.975,179.664,5.989,149.173
C01351=1161.389,-17.609,-45.963,179.661,5.988,149.173
C01352=1161.393,-17.859,-45.950,179.659,5.988,149.174
C01353=1161.398,-18.109,-45.938,179.656,5.987,149.174
C01354=1161.404,-18.358,-45.924,179.654,5.986,149.175
C01355=1161.409,-18.608,-45.912,179.651,5.986,149.176
C01356=1161.415,-18.857,-45.900,179.649,5.985,149.176
C01357=1161.420,-19.107,-45.887,179.647,5.985,149.177
C01358=1161.424,-19.357,-45.874,179.644,5.984,149.177
C01359=1161.429,-19.606,-45.862,179.642,5.983,149.178
C01360=1161.435,-19.856,-45.850,179.640,5.983,149.178
C01361=1161.440,-20.105,-45.837,179.637,5.982,149.179
C01362=1161.445,-20.355,-45.825,179.634,5.982,149.180
C01363=1161.450,-20.605,-45.812,179.632,5.981,149.180
C01364=1161.456,-20.855,-45.799,179.629,5.980,149.181
C01365=1161.461,-21.104,-45.787,179.627,5.980,149.181
C01366=1161.466,-21.354,-45.774,179.625,5.979,149.182
C01367=1161.471,-21.604,-45.762,179.622,5.978,149.183
C01368=1161.477,-21.853,-45.750,179.620,5.978,149.183
C01369=1161.482,-22.102,-45.737,179.618,5.977,149.184
C01370=1161.487,-22.353,-45.725,179.615,5.977,149.184
C01371=1161.492,-22.602,-45.712,179.612,5.976,149.185
C01372=1161.497,-22.851,-45.699,179.610,5.976,149.186
C01373=1161.502,-23.101,-45.688,179.607,5.975,149.186
C01374=1161.507,-23.351,-45.675,179.605,5.974,149.187
C01375=1161.512,-23.600,-45.662,179.603,5.974,149.187
C01376=1161.518,-23.870,-45.649,179.600,5.973,149.188
C01377=1161.524,-24.140,-45.636,179.598,5.973,149.189
C01378=1161.529,-24.410,-45.623,179.595,5.972,149.189
C01379=1161.535,-24.680,-45.610,179.592,5.972,149.190
C01380=1161.540,-24.930,-45.597,179.590,5.971,149.190
C01381=1161.545,-25.179,-45.584,179.588,5.971,149.191
C01382=1161.550,-25.429,-45.572,179.585,5.970,149.192
C01383=1161.556,-25.678,-45.560,179.583,5.969,149.192
C01384=1161.561,-25.928,-45.548,179.581,5.968,149.193
C01385=1161.566,-26.178,-45.535,179.578,5.968,149.194
C01386=1161.572,-26.427,-45.524,179.575,5.968,149.194
C01387=1161.577,-26.677,-45.511,179.573,5.967,149.195
C01388=1161.581,-26.927,-45.499,179.570,5.966,149.195
C01389=1161.587,-27.177,-45.486,179.568,5.966,149.196
C01390=1161.592,-27.427,-45.474,179.566,5.965,149.197
C01391=1161.596,-27.676,-45.462,179.563,5.964,149.197
C01392=1161.602,-27.926,-45.450,179.561,5.965,149.198
C01393=1161.607,-28.175,-45.438,179.559,5.964,149.198
C01394=1161.612,-28.425,-45.426,179.556,5.963,149.199
C01395=1161.618,-28.674,-45.413,179.554,5.963,149.199
C01396=1161.623,-28.924,-45.401,179.552,5.962,149.200
C01397=1161.628,-29.173,-45.389,179.549,5.962,149.201
C01398=1161.634,-29.423,-45.377,179.547,5.961,149.201
C01399=1161.639,-29.673,-45.365,179.544,5.961,149.202
C01400=1161.643,-29.922,-45.353,179.542,5.960,149.202
C01401=1161.649,-30.172,-45.341,179.539,5.959,149.203
C01402=1161.654,-30.422,-45.328,179.537,5.959,149.204
C01403=1161.659,-30.672,-45.317,179.534,5.958,149.204
C01404=1161.664,-30.921,-45.304,179.532,5.957,149.205
C01405=1161.670,-31.171,-45.292,179.530,5.958,149.205
C01406=1161.675,-31.420,-45.281,179.528,5.957,149.206
C01407=1161.680,-31.670,-45.268,179.525,5.956,149.207
C01408=1161.685,-31.920,-45.256,179.523,5.956,149.207
C01409=1161.691,-32.170,-45.244,179.520,5.955,149.208
C01410=1161.696,-32.419,-45.232,179.518,5.955,149.208
C01411=1161.700,-32.669,-45.221,179.516,5.954,149.209
C01412=1161.706,-32.918,-45.209,179.513,5.954,149.210
C01413=1161.711,-33.168,-45.196,179.511,5.953,149.210
C01414=1161.716,-33.418,-45.184,179.508,5.952,149.211
C01415=1161.722,-33.668,-45.172,179.506,5.952,149.211
C01416=1161.726,-33.917,-45.160,179.504,5.952,149.212
C01417=1161.732,-34.167,-45.148,179.502,5.951,149.212
C01418=1161.737,-34.417,-45.136,179.499,5.951,149.213
C01419=1161.742,-34.666,-45.125,179.497,5.950,149.214
C01420=1161.747,-34.915,-45.113,179.494,5.949,149.214
C01421=1161.752,-35.165,-45.101,179.492,5.949,149.215
C01422=1161.758,-35.415,-45.089,179.489,5.948,149.216
C01423=1161.763,-35.665,-45.077,179.487,5.948,149.216
C01424=1161.768,-35.914,-45.065,179.484,5.947,149.217
C01425=1161.774,-36.164,-45.053,179.482,5.947,149.217
C01426=1161.779,-36.413,-45.042,179.480,5.947,149.218
C01427=1161.784,-36.663,-45.030,179.478,5.946,149.219
C01428=1161.789,-36.913,-45.018,179.475,5.945,149.219
C01429=1161.794,-37.162,-45.006,179.473,5.945,149.220
C01430=1161.800,-37.412,-44.994,179.471,5.944,149.220
C01431=1161.804,-37.662,-44.983,179.468,5.944,149.221
C01432=1161.810,-37.912,-44.971,179.466,5.943,149.221
C01433=1161.815,-38.162,-44.959,179.463,5.942,149.222
C01434=1161.820,-38.411,-44.948,179.461,5.943,149.223
C01435=1161.825,-38.661,-44.935,179.459,5.942,149.223
C01436=1161.831,-38.910,-44.923,179.456,5.942,149.224
C01437=1161.836,-39.160,-44.912,179.454,5.941,149.224
C01438=1161.841,-39.410,-44.900,179.451,5.940,149.225
C01439=1161.847,-39.659,-44.888,179.449,5.940,149.226
C01440=1161.851,-39.909,-44.877,179.446,5.939,149.226
C01441=1161.857,-40.159,-44.865,179.444,5.938,149.227
C01442=1161.862,-40.409,-44.853,179.442,5.939,149.227
C01443=1161.867,-40.658,-44.842,179.440,5.938,149.228
C01444=1161.873,-40.907,-44.830,179.437,5.938,149.229
C01445=1161.878,-41.157,-44.818,179.435,5.937,149.229
C01446=1161.883,-41.407,-44.807,179.432,5.936,149.230
C01447=1161.888,-41.657,-44.795,179.430,5.936,149.230
C01448=1161.893,-41.906,-44.783,179.428,5.935,149.231
C01449=1161.898,-42.156,-44.772,179.426,5.936,149.232
C01450=1161.904,-42.405,-44.760,179.423,5.935,149.232
C01451=1161.909,-42.655,-44.749,179.421,5.934,149.233
C01452=1161.914,-42.905,-44.737,179.419,5.933,149.233
C01453=1161.919,-43.155,-44.726,179.416,5.933,149.234
C01454=1161.924,-43.405,-44.714,179.414,5.932,149.235
C01455=1161.929,-43.654,-44.702,179.411,5.932,149.235
C01456=1161.935,-43.903,-44.691,179.409,5.932,149.236
C01457=1161.941,-44.153,-44.679,179.407,5.931,149.236
C01458=1161.945,-44.403,-44.668,179.405,5.931,149.237
C01459=1161.951,-44.653,-44.656,179.402,5.930,149.238
C01460=1161.955,-44.903,-44.644,179.400,5.929,149.238
C01461=1161.961,-45.152,-44.633,179.397,5.929,149.239
C01462=1161.966,-45.401,-44.622,179.395,5.929,149.239
C01463=1161.972,-45.651,-44.610,179.393,5.929,149.240
C01464=1161.976,-45.901,-44.599,179.391,5.928,149.240
C01465=1161.982,-46.152,-44.587,179.388,5.927,149.241
C01466=1161.987,-46.401,-44.576,179.386,5.927,149.242
C01467=1161.993,-46.650,-44.565,179.383,5.926,149.242
C01468=1161.997,-46.900,-44.553,179.381,5.927,149.243
C01469=1162.003,-47.150,-44.541,179.379,5.926,149.243
C01470=1162.008,-47.399,-44.530,179.376,5.925,149.244
C01471=1162.014,-47.649,-44.519,179.374,5.925,149.245
C01472=1162.018,-47.898,-44.507,179.371,5.924,149.245
C01473=1162.024,-48.149,-44.496,179.369,5.923,149.246
C01474=1162.029,-48.398,-44.485,179.367,5.924,149.247
C01475=1162.035,-48.648,-44.473,179.365,5.923,149.247
C01476=1162.039,-48.898,-44.462,179.362,5.923,149.248
C01477=1162.044,-49.147,-44.451,179.360,5.922,149.248
C01478=1162.050,-49.396,-44.439,179.357,5.921,149.249
C01479=1162.055,-49.647,-44.429,179.355,5.921,149.249
C01480=1162.060,-49.917,-44.416,179.352,5.920,149.250
C01481=1162.067,-50.187,-44.404,179.350,5.920,149.251
C01482=1162.072,-50.458,-44.391,179.348,5.920,149.251
C01483=1162.078,-50.729,-44.379,179.346,5.919,149.252
C01484=1162.083,-50.978,-44.368,179.343,5.919,149.253
C01485=1162.089,-51.228,-44.356,179.341,5.918,149.253
C01486=1162.093,-51.478,-44.345,179.338,5.918,149.254
C01487=1162.098,-51.727,-44.334,179.336,5.917,149.254
C01488=1162.104,-51.977,-44.323,179.334,5.917,149.255
C01489=1162.109,-52.227,-44.312,179.332,5.916,149.256
C01490=1162.114,-52.477,-44.300,179.329,5.916,149.256
C01491=1162.120,-52.726,-44.290,179.327,5.915,149.257
C01492=1162.125,-52.976,-44.278,179.324,5.915,149.257
C01493=1162.130,-53.226,-44.266,179.322,5.914,149.258
C01494=1162.136,-53.475,-44.256,179.320,5.914,149.259
C01495=1162.141,-53.725,-44.245,179.318,5.914,149.259
C01496=1162.146,-53.975,-44.233,179.315,5.913,149.260
C01497=1162.151,-54.224,-44.222,179.313,5.912,149.260
C01498=1162.156,-54.474,-44.212,179.311,5.913,149.261
C01499=1162.162,-54.724,-44.200,179.309,5.912,149.261
C01500=1162.167,-54.973,-44.189,179.306,5.912,149.262
C01501=1162.172,-55.223,-44.178,179.304,5.911,149.263
C01502=1162.177,-55.473,-44.167,179.301,5.910,149.263
C01503=1162.183,-55.722,-44.155,179.299,5.910,149.264
C01504=1162.188,-55.972,-44.145,179.297,5.910,149.264
C01505=1162.192,-56.222,-44.134,179.295,5.909,149.265
C01506=1162.199,-56.472,-44.123,179.292,5.909,149.266
C01507=1162.203,-56.721,-44.111,179.290,5.908,149.266
C01508=1162.208,-56.971,-44.100,179.288,5.908,149.267
C01509=1162.214,-57.221,-44.090,179.285,5.908,149.267
C01510=1162.219,-57.471,-44.078,179.283,5.907,149.268
C01511=1162.225,-57.720,-44.068,179.281,5.906,149.269
C01512=1162.229,-57.970,-44.057,179.278,5.906,149.269
C01513=1162.234,-58.220,-44.046,179.276,5.906,149.270
C01514=1162.240,-58.469,-44.034,179.274,5.906,149.270
C01515=1162.245,-58.719,-44.023,179.271,5.905,149.271
C01516=1162.251,-58.968,-44.013,179.269,5.904,149.272
C01517=1162.255,-59.218,-44.002,179.267,5.904,149.272
C01518=1162.260,-59.468,-43.991,179.265,5.904,149.273
C01519=1162.266,-59.717,-43.980,179.262,5.903,149.273
C01520=1162.271,-59.968,-43.969,179.260,5.903,149.274
C01521=1162.277,-60.217,-43.958,179.258,5.903,149.274
C01522=1162.282,-60.467,-43.948,179.255,5.902,149.275
C01523=1162.286,-60.717,-43.936,179.253,5.902,149.276
C01524=1162.293,-60.966,-43.925,179.251,5.901,149.276
C01525=1162.297,-61.216,-43.914,179.248,5.900,149.277
C01526=1162.303,-61.466,-43.904,179.246,5.901,149.277
C01527=1162.308,-61.715,-43.893,179.244,5.900,149.278
C01528=1162.313,-61.965,-43.882,179.241,5.900,149.279
C01529=1162.319,-62.215,-43.871,179.239,5.899,149.279
C01530=1162.324,-62.465,-43.860,179.237,5.899,149.280
C01531=1162.329,-62.714,-43.850,179.235,5.899,149.280
C01532=1162.334,-62.964,-43.838,179.232,5.898,149.281
C01533=1162.340,-63.214,-43.828,179.230,5.897,149.282
C01534=1162.344,-63.463,-43.817,179.228,5.898,149.282
C01535=1162.350,-63.713,-43.807,179.226,5.897,149.283
C01536=1162.355,-63.963,-43.796,179.223,5.897,149.283
C01537=1162.361,-64.212,-43.785,179.221,5.896,149.284
C01538=1162.366,-64.463,-43.774,179.219,5.896,149.285
C01539=1162.372,-64.712,-43.764,179.217,5.895,149.285
C01540=1162.376,-64.962,-43.753,179.214,5.895,149.286
C01541=1162.382,-65.211,-43.742,179.212,5.894,149.286
C01542=1162.387,-65.461,-43.732,179.210,5.895,149.287
C01543=1162.392,-65.710,-43.721,179.208,5.894,149.287
C01544=1162.397,-65.961,-43.710,179.205,5.893,149.288
C01545=1162.403,-66.210,-43.700,179.203,5.893,149.289
C01546=1162.407,-66.460,-43.689,179.201,5.893,149.289
C01547=1162.414,-66.710,-43.678,179.199,5.892,149.290
C01548=1162.419,-66.960,-43.667,179.196,5.891,149.290
C01549=1162.424,-67.209,-43.657,179.194,5.892,149.291
C01550=1162.429,-67.459,-43.646,179.192,5.891,149.291
C01551=1162.435,-67.709,-43.636,179.189,5.891,149.292
C01552=1162.439,-67.958,-43.624,179.187,5.890,149.293
C01553=1162.445,-68.208,-43.614,179.185,5.890,149.293
C01554=1162.450,-68.458,-43.604,179.183,5.889,149.294
C01555=1162.456,-68.708,-43.593,179.180,5.889,149.295
C01556=1162.460,-68.957,-43.582,179.178,5.888,149.295
C01557=1162.466,-69.207,-43.572,179.176,5.889,149.296
C01558=1162.471,-69.457,-43.561,179.174,5.888,149.296
C01559=1162.476,-69.707,-43.551,179.171,5.887,149.297
C01560=1162.482,-69.956,-43.541,179.170,5.887,149.297
C01561=1162.487,-70.206,-43.530,179.167,5.887,149.298
C01562=1162.492,-70.455,-43.519,179.165,5.886,149.299
C01563=1162.497,-70.705,-43.509,179.162,5.886,149.299
C01564=1162.503,-70.955,-43.499,179.160,5.886,149.300
C01565=1162.508,-71.205,-43.488,179.158,5.885,149.300
C01566=1162.513,-71.454,-43.477,179.156,5.885,149.301
C01567=1162.519,-71.704,-43.467,179.153,5.884,149.301
C01568=1162.524,-71.954,-43.456,179.151,5.884,149.302
C01569=1162.529,-72.204,-43.446,179.149,5.884,149.303
C01570=1162.534,-72.454,-43.436,179.146,5.883,149.303
C01571=1162.540,-72.703,-43.425,179.145,5.883,149.304
C01572=1162.546,-72.953,-43.415,179.142,5.883,149.305
C01573=1162.550,-73.202,-43.404,179.140,5.882,149.305
C01574=1162.556,-73.452,-43.394,179.138,5.882,149.306
C01575=1162.561,-73.702,-43.383,179.136,5.882,149.306
C01576=1162.566,-73.951,-43.374,179.133,5.881,149.307
C01577=1162.571,-74.201,-43.363,179.131,5.880,149.307
C01578=1162.576,-74.451,-43.353,179.129,5.880,149.308
C01579=1162.582,-74.701,-43.343,179.127,5.880,149.309
C01580=1162.588,-74.950,-43.332,179.124,5.879,149.309
C01581=1162.593,-75.201,-43.322,179.122,5.880,149.310
C01582=1162.598,-75.450,-43.312,179.120,5.879,149.310
C01583=1162.603,-75.700,-43.301,179.117,5.879,149.311
C01584=1162.609,-75.970,-43.290,179.115,5.878,149.311
C01585=1162.615,-76.242,-43.278,179.113,5.878,149.312
C01586=1162.620,-76.513,-43.267,179.111,5.878,149.313
C01587=1162.626,-76.784,-43.256,179.108,5.877,149.313
C01588=1162.631,-77.034,-43.245,179.106,5.877,149.314
C01589=1162.637,-77.284,-43.235,179.103,5.876,149.315
C01590=1162.642,-77.534,-43.225,179.101,5.876,149.315
C01591=1162.647,-77.783,-43.215,179.099,5.875,149.316
C01592=1162.652,-78.033,-43.205,179.097,5.875,149.316
C01593=1162.658,-78.283,-43.195,179.095,5.875,149.317
C01594=1162.663,-78.533,-43.184,179.093,5.874,149.317
C01595=1162.668,-78.782,-43.174,179.090,5.874,149.318
C01596=1162.674,-79.032,-43.164,179.088,5.874,149.319
C01597=1162.679,-79.282,-43.154,179.086,5.874,149.319
C01598=1162.684,-79.532,-43.144,179.084,5.873,149.320
C01599=1162.690,-79.782,-43.134,179.082,5.873,149.321
C01600=1162.695,-80.031,-43.124,179.079,5.872,149.321
C01601=1162.700,-80.281,-43.113,179.077,5.872,149.322
C01602=1162.705,-80.531,-43.104,179.075,5.872,149.322
C01603=1162.711,-80.780,-43.093,179.073,5.871,149.323
C01604=1162.716,-81.030,-43.083,179.070,5.871,149.323
C01605=1162.721,-81.280,-43.073,179.069,5.871,149.324
C01606=1162.727,-81.529,-43.062,179.066,5.870,149.325
C01607=1162.732,-81.779,-43.053,179.064,5.870,149.325
C01608=1162.737,-82.030,-43.043,179.062,5.870,149.326
C01609=1162.743,-82.279,-43.033,179.060,5.869,149.326
C01610=1162.748,-82.529,-43.022,179.057,5.869,149.327
C01611=1162.753,-82.779,-43.012,179.055,5.869,149.327
C01612=1162.758,-83.028,-43.002,179.053,5.868,149.328
C01613=1162.764,-83.278,-42.992,179.050,5.868,149.329
C01614=1162.770,-83.527,-42.982,179.049,5.868,149.329
C01615=1162.774,-83.778,-42.973,179.046,5.867,149.330
C01616=1162.780,-84.027,-42.962,179.044,5.867,149.330
C01617=1162.785,-84.277,-42.952,179.042,5.867,149.331
C01618=1162.790,-84.526,-42.943,179.040,5.866,149.331
C01619=1162.795,-84.776,-42.932,179.037,5.865,149.332
C01620=1162.801,-85.026,-42.922,179.035,5.866,149.333
C01621=1162.806,-85.276,-42.913,179.033,5.865,149.333
C01622=1162.811,-85.525,-42.903,179.031,5.865,149.334
C01623=1162.816,-85.775,-42.892,179.029,5.865,149.334
C01624=1162.821,-86.025,-42.882,179.027,5.864,149.335
C01625=1162.827,-86.275,-42.873,179.024,5.864,149.336
C01626=1162.833,-86.524,-42.863,179.022,5.864,149.336
C01627=1162.838,-86.774,-42.853,179.020,5.863,149.337
C01628=1162.843,-87.024,-42.843,179.018,5.862,149.337
C01629=1162.849,-87.274,-42.833,179.016,5.862,149.338
C01630=1162.853,-87.523,-42.823,179.013,5.862,149.338
C01631=1162.859,-87.773,-42.813,179.012,5.862,149.339
C01632=1162.864,-88.024,-42.803,179.009,5.862,149.340
C01633=1162.869,-88.273,-42.794,179.007,5.861,149.340
C01634=1162.875,-88.522,-42.784,179.005,5.861,149.341
C01635=1162.880,-88.772,-42.773,179.003,5.861,149.341
C01636=1162.886,-89.022,-42.764,179.000,5.860,149.342
C01637=1162.891,-89.271,-42.754,178.998,5.860,149.342
C01638=1162.895,-89.521,-42.744,178.996,5.859,149.343
C01639=1162.901,-89.771,-42.735,178.993,5.859,149.344
C01640=1162.907,-90.021,-42.725,178.992,5.859,149.344
C01641=1162.912,-90.270,-42.715,178.990,5.858,149.345
C01642=1162.918,-90.520,-42.706,178.988,5.859,149.345
C01643=1162.922,-90.770,-42.696,178.985,5.858,149.346
C01644=1162.928,-91.021,-42.686,178.983,5.858,149.347
C01645=1162.933,-91.270,-42.676,178.981,5.858,149.347
C01646=1162.938,-91.519,-42.666,178.979,5.857,149.348
C01647=1162.944,-91.769,-42.657,178.976,5.856,149.348
C01648=1162.949,-92.019,-42.647,178.975,5.856,149.349
C01649=1162.955,-92.268,-42.637,178.972,5.856,149.349
C01650=1162.959,-92.519,-42.628,178.970,5.856,149.350
C01651=1162.965,-92.768,-42.617,178.968,5.855,149.350
C01652=1162.970,-93.018,-42.609,178.966,5.855,149.351
C01653=1162.976,-93.268,-42.598,178.964,5.855,149.352
C01654=1162.981,-93.518,-42.589,178.961,5.855,149.352
C01655=1162.986,-93.767,-42.579,178.959,5.854,149.353
C01656=1162.991,-94.016,-42.570,178.957,5.854,149.353
C01657=1162.997,-94.266,-42.560,178.955,5.853,149.354
C01658=1163.001,-94.516,-42.550,178.953,5.853,149.354
C01659=1163.007,-94.767,-42.541,178.951,5.853,149.355
C01660=1163.013,-95.016,-42.530,178.948,5.852,149.356
C01661=1163.018,-95.266,-42.522,178.947,5.852,149.356
C01662=1163.024,-95.516,-42.511,178.944,5.852,149.357
C01663=1163.029,-95.765,-42.502,178.942,5.852,149.357
C01664=1163.034,-96.015,-42.493,178.940,5.851,149.358
C01665=1163.040,-96.265,-42.483,178.938,5.851,149.359
C01666=1163.044,-96.514,-42.474,178.936,5.851,149.359
C01667=1163.050,-96.764,-42.464,178.934,5.850,149.360
C01668=1163.055,-97.013,-42.455,178.932,5.850,149.360
C01669=1163.061,-97.264,-42.445,178.930,5.850,149.361
C01670=1163.066,-97.514,-42.436,178.927,5.849,149.361
C01671=1163.071,-97.764,-42.426,178.925,5.849,149.362
C01672=1163.076,-98.014,-42.417,178.923,5.849,149.362
C01673=1163.082,-98.263,-42.407,178.920,5.848,149.363
C01674=1163.087,-98.513,-42.398,178.919,5.848,149.364
C01675=1163.093,-98.762,-42.387,178.917,5.847,149.364
C01676=1163.098,-99.012,-42.379,178.915,5.848,149.365
C01677=1163.103,-99.262,-42.370,178.912,5.847,149.365
C01678=1163.109,-99.512,-42.359,178.910,5.847,149.366
C01679=1163.114,-99.762,-42.351,178.908,5.847,149.366
C01680=1163.120,-100.011,-42.340,178.906,5.846,149.367
C01681=1163.125,-100.261,-42.331,178.904,5.846,149.368
C01682=1163.130,-100.511,-42.322,178.902,5.846,149.368
C01683=1163.135,-100.760,-42.312,178.900,5.846,149.369
C01684=1163.141,-101.010,-42.303,178.897,5.845,149.369
C01685=1163.147,-101.260,-42.294,178.895,5.844,149.370
C01686=1163.151,-101.510,-42.284,178.894,5.845,149.370
C01687=1163.157,-101.759,-42.275,178.891,5.844,149.371
C01688=1163.162,-102.031,-42.265,178.889,5.843,149.372
C01689=1163.168,-102.304,-42.254,178.887,5.844,149.372
C01690=1163.174,-102.576,-42.244,178.884,5.843,149.373
C01691=1163.180,-102.847,-42.234,178.882,5.843,149.373
C01692=1163.185,-103.097,-42.225,178.880,5.843,149.374
C01693=1163.191,-103.347,-42.216,178.877,5.842,149.375
C01694=1163.196,-103.596,-42.206,178.876,5.842,149.375
C01695=1163.201,-103.846,-42.197,178.874,5.842,149.376
C01696=1163.207,-104.096,-42.188,178.871,5.841,149.376
C01697=1163.212,-104.346,-42.179,178.869,5.841,149.377
C01698=1163.217,-104.595,-42.169,178.867,5.840,149.377
C01699=1163.223,-104.845,-42.160,178.865,5.841,149.378
C01700=1163.228,-105.095,-42.151,178.863,5.840,149.378
C01701=1163.233,-105.345,-42.142,178.861,5.840,149.379
C01702=1163.239,-105.594,-42.132,178.859,5.840,149.380
C01703=1163.244,-105.844,-42.123,178.856,5.839,149.380
C01704=1163.249,-106.094,-42.114,178.855,5.839,149.381
C01705=1163.254,-106.344,-42.105,178.852,5.839,149.381
C01706=1163.260,-106.594,-42.095,178.851,5.839,149.382
C01707=1163.265,-106.843,-42.086,178.848,5.838,149.382
C01708=1163.270,-107.093,-42.077,178.846,5.838,149.383
C01709=1163.275,-107.343,-42.068,178.844,5.838,149.384
C01710=1163.281,-107.593,-42.059,178.842,5.837,149.384
C01711=1163.286,-107.843,-42.049,178.840,5.837,149.385
C01712=1163.291,-108.092,-42.040,178.838,5.836,149.385
C01713=1163.296,-108.342,-42.031,178.836,5.836,149.386
C01714=1163.302,-108.592,-42.022,178.833,5.836,149.386
C01715=1163.308,-108.842,-42.013,178.832,5.836,149.387
C01716=1163.313,-109.092,-42.004,178.830,5.835,149.387
C01717=1163.318,-109.341,-41.996,178.828,5.836,149.388
C01718=1163.324,-109.591,-41.985,178.825,5.835,149.389
C01719=1163.329,-109.841,-41.976,178.823,5.834,149.389
C01720=1163.334,-110.090,-41.968,178.821,5.835,149.390
C01721=1163.340,-110.340,-41.959,178.819,5.834,149.390
C01722=1163.345,-110.590,-41.950,178.817,5.834,149.391
C01723=1163.351,-110.840,-41.940,178.815,5.834,149.391
C01724=1163.356,-111.090,-41.931,178.813,5.834,149.392
C01725=1163.361,-111.340,-41.922,178.811,5.833,149.392
C01726=1163.366,-111.590,-41.914,178.809,5.833,149.393
C01727=1163.372,-111.838,-41.904,178.806,5.832,149.394
C01728=1163.377,-112.089,-41.895,178.805,5.833,149.394
C01729=1163.383,-112.338,-41.886,178.802,5.832,149.395
C01730=1163.388,-112.588,-41.877,178.800,5.831,149.395
C01731=1163.393,-112.838,-41.868,178.798,5.831,149.396
C01732=1163.398,-113.088,-41.859,178.796,5.831,149.396
C01733=1163.403,-113.338,-41.850,178.794,5.831,149.397
C01734=1163.409,-113.588,-41.841,178.792,5.830,149.398
C01735=1163.415,-113.837,-41.832,178.790,5.830,149.398
C01736=1163.420,-114.087,-41.823,178.788,5.830,149.399
C01737=1163.425,-114.337,-41.814,178.786,5.830,149.399
C01738=1163.430,-114.587,-41.806,178.784,5.829,149.400
C01739=1163.436,-114.837,-41.797,178.782,5.829,149.400
C01740=1163.441,-115.086,-41.788,178.780,5.829,149.401
C01741=1163.447,-115.337,-41.778,178.778,5.829,149.401
C01742=1163.452,-115.586,-41.770,178.776,5.828,149.402
C01743=1163.458,-115.836,-41.761,178.773,5.828,149.403
C01744=1163.463,-116.085,-41.752,178.772,5.828,149.403
C01745=1163.468,-116.335,-41.743,178.769,5.827,149.404
C01746=1163.473,-116.585,-41.734,178.767,5.827,149.404
C01747=1163.479,-116.834,-41.726,178.765,5.827,149.405
C01748=1163.484,-117.084,-41.717,178.763,5.827,149.405
C01749=1163.489,-117.334,-41.708,178.761,5.826,149.406
C01750=1163.494,-117.584,-41.699,178.759,5.826,149.406
C01751=1163.500,-117.834,-41.691,178.757,5.826,149.407
C01752=1163.506,-118.084,-41.681,178.755,5.826,149.407
C01753=1163.512,-118.334,-41.673,178.753,5.825,149.408
C01754=1163.517,-118.583,-41.664,178.751,5.825,149.409
C01755=1163.522,-118.833,-41.655,178.749,5.825,149.409
C01756=1163.527,-119.083,-41.646,178.747,5.825,149.410
C01757=1163.532,-119.333,-41.637,178.745,5.824,149.410
C01758=1163.538,-119.582,-41.629,178.743,5.824,149.411
C01759=1163.543,-119.832,-41.620,178.741,5.824,149.411
C01760=1163.548,-120.082,-41.611,178.739,5.824,149.412
C01761=1163.554,-120.332,-41.603,178.737,5.823,149.412
C01762=1163.560,-120.582,-41.594,178.735,5.823,149.413
C01763=1163.565,-120.831,-41.585,178.733,5.822,149.413
C01764=1163.570,-121.081,-41.576,178.731,5.823,149.414
C01765=1163.575,-121.331,-41.567,178.729,5.822,149.415
C01766=1163.580,-121.581,-41.559,178.727,5.822,149.415
C01767=1163.586,-121.831,-41.551,178.725,5.821,149.416
C01768=1163.591,-122.081,-41.542,178.723,5.821,149.416
C01769=1163.597,-122.330,-41.533,178.720,5.821,149.417
C01770=1163.602,-122.580,-41.524,178.718,5.820,149.417
C01771=1163.608,-122.829,-41.515,178.717,5.820,149.418
C01772=1163.613,-123.080,-41.507,178.714,5.820,149.418
C01773=1163.618,-123.330,-41.498,178.712,5.820,149.419
C01774=1163.623,-123.580,-41.489,178.710,5.819,149.419
C01775=1163.629,-123.829,-41.481,178.709,5.819,149.420
C01776=1163.634,-124.079,-41.472,178.706,5.819,149.420
C01777=1163.640,-124.329,-41.464,178.704,5.819,149.421
C01778=1163.646,-124.578,-41.455,178.702,5.818,149.422
C01779=1163.650,-124.828,-41.447,178.701,5.818,149.422
C01780=1163.655,-125.078,-41.438,178.698,5.817,149.423
C01781=1163.661,-125.328,-41.430,178.696,5.818,149.423
C01782=1163.666,-125.577,-41.421,178.694,5.817,149.424
C01783=1163.672,-125.827,-41.413,178.692,5.817,149.424
C01784=1163.677,-126.078,-41.404,178.691,5.817,149.425
C01785=1163.683,-126.327,-41.396,178.688,5.817,149.426
C01786=1163.688,-126.577,-41.387,178.687,5.817,149.426
C01787=1163.693,-126.826,-41.378,178.684,5.816,149.427
C01788=1163.699,-127.077,-41.370,178.683,5.816,149.427
C01789=1163.704,-127.326,-41.361,178.680,5.816,149.428
C01790=1163.710,-127.576,-41.352,178.679,5.816,149.428
C01791=1163.714,-127.826,-41.345,178.676,5.815,149.429
C01792=1163.293,-127.837,-41.386,178.672,5.818,149.431
C01793=1163.288,-127.587,-41.394,178.675,5.819,149.430
C01794=1163.283,-127.337,-41.403,178.677,5.819,149.429
C01795=1163.277,-127.088,-41.412,178.679,5.819,149.429
C01796=1163.272,-126.838,-41.420,178.680,5.819,149.428
C01797=1163.266,-126.587,-41.429,178.683,5.820,149.428
C01798=1163.262,-126.338,-41.437,178.684,5.820,149.427
C01799=1163.256,-126.089,-41.446,178.687,5.820,149.427
C01800=1163.251,-125.838,-41.454,178.689,5.820,149.426
C01801=1163.246,-125.588,-41.463,178.691,5.821,149.426
C01802=1163.240,-125.339,-41.471,178.692,5.821,149.425
C01803=1163.234,-125.089,-41.479,178.695,5.822,149.424
C01804=1163.229,-124.839,-41.488,178.697,5.822,149.424
C01805=1163.224,-124.589,-41.497,178.699,5.822,149.423
C01806=1163.218,-124.340,-41.506,178.700,5.822,149.423
C01807=1163.213,-124.089,-41.514,178.703,5.823,149.422
C01808=1163.208,-123.840,-41.523,178.705,5.823,149.422
C01809=1163.202,-123.590,-41.531,178.707,5.823,149.421
C01810=1163.197,-123.341,-41.540,178.709,5.823,149.421
C01811=1163.191,-123.091,-41.549,178.711,5.824,149.420
C01812=1163.186,-122.840,-41.557,178.713,5.824,149.420
C01813=1163.180,-122.591,-41.566,178.715,5.824,149.419
C01814=1163.175,-122.341,-41.575,178.717,5.824,149.419
C01815=1163.170,-122.091,-41.584,178.719,5.825,149.418
C01816=1163.165,-121.842,-41.592,178.721,5.825,149.417
C01817=1163.159,-121.592,-41.600,178.723,5.825,149.417
C01818=1163.154,-121.342,-41.609,178.725,5.825,149.416
C01819=1163.148,-121.092,-41.618,178.727,5.826,149.416
C01820=1163.143,-120.842,-41.627,178.729,5.826,149.415
C01821=1163.138,-120.592,-41.636,178.731,5.826,149.415
C01822=1163.132,-120.343,-41.644,178.733,5.826,149.414
C01823=1163.127,-120.093,-41.653,178.735,5.827,149.414
C01824=1163.122,-119.843,-41.661,178.737,5.827,149.413
C01825=1163.116,-119.593,-41.670,178.739,5.828,149.413
C01826=1163.111,-119.344,-41.679,178.741,5.828,149.412
